// TwinCAT 3 PLC project PLC_Tool_Magazine_8xx
// ProgramVersion: 3.1.4026.20
// libraries:
//   Tc2_Drive, * (Beckhoff Automation GmbH)
//   Tc2_Math, * (Beckhoff Automation GmbH)
//   Tc2_MC2, * (Beckhoff Automation GmbH)
//   Tc2_MC2_Drive, * (Beckhoff Automation GmbH)
//   Tc2_Standard, * (Beckhoff Automation GmbH)
//   Tc2_System, * (Beckhoff Automation GmbH)
//   Tc2_Utilities, * (Beckhoff Automation GmbH)
//   Tc3_EventLogger, * (Beckhoff Automation GmbH)
//   Tc3_IoLink, * (Beckhoff Automation GmbH)
//   Tc3_Module, * (Beckhoff Automation GmbH)
// project tree:
//   01_General %28MAIN%29/01_DUTs/01_ENUM/ ENUM_VarType.TcDUT (not stored)
//   01_General %28MAIN%29/01_DUTs/02_ST/ ST_Array_Data.TcDUT (not stored), ST_Miscellaneous.TcDUT (not stored), ST_Pointer_Data.TcDUT (not stored)
//   01_General %28MAIN%29/02_GVLs/ GV_General.TcGVL (not stored), GV_IO.TcGVL (not stored)
//   01_General %28MAIN%29/03_POUs/01_PRGs/ PRG_Backup.TcPOU (not stored), PRG_FirstCycle.TcPOU (not stored), PRG_Main.TcPOU (not stored), PRG_SavePersistentData.TcPOU (not stored)
//   01_General %28MAIN%29/03_POUs/02_FBs/ FB_ArrayToolLocation_Reverse.TcPOU (not stored), FB_BackupExport.TcPOU (not stored), FB_BackupImport.TcPOU (not stored), FB_Blink.TcPOU (not stored)
//   02_Events/01_DUTs/02_ST/ ST_Alarm.TcDUT, ST_Event_Group.TcDUT, ST_Message.TcDUT
//   02_Events/02_GVLs/ GV_Events.TcGVL
//   02_Events/03_POUs/02_FBs/ FB_Event_Group_Number_Assignement.TcPOU, FB_Event_HMI.TcPOU, FB_Init_Call_Events.TcPOU, FB_Init_Events.TcPOU
//   03_Operating_Mode/01_DUTs/01_ENUM/ ENUM_OpMode.TcDUT
//   03_Operating_Mode/02_GVLs/ GV_OpMode.TcGVL
//   03_Operating_Mode/03_POUs/01_PRGs/ PRG_OpMode.TcPOU
//   04_Lamps_Lights/03_POUs/01_PRGs/ PRG_Lamps_Lights.TcPOU
//   05_Fans/01_DUTs/01_ENUM/ ENUM_Fan_Type.TcDUT
//   05_Fans/01_DUTs/02_ST/ ST_Fan.TcDUT
//   05_Fans/02_GVLs/ GV_Fans.TcGVL
//   05_Fans/03_POUs/01_PRGs/ PRG_Fans.TcPOU
//   05_Fans/03_POUs/02_FBs/ FB_Fan.TcPOU
//   06_Doors/01_DUTs/01_ENUM/ ENUM_Door_Type.TcDUT
//   06_Doors/01_DUTs/02_ST/ ST_Door.TcDUT
//   06_Doors/02_GVLs/ GV_Doors.TcGVL
//   06_Doors/03_POUs/01_PRGs/ PRG_Doors.TcPOU
//   06_Doors/03_POUs/02_FBs/ FB_Door.TcPOU
//   07_Cyltronic/01_DUTs/01_ENUM/ ENUM_Cyltronic_Type.TcDUT, teCTCBrakeMode.TcTLEO, teCTCConfigStep.TcDUT, teCTCDeviceStatus.TcTLEO, teCTCEvent.TcTLEO, teCTCGDSStep.TcDUT, teCTCHomeMode.TcTLEO, teCTCStep.TcTLEO, teCTCWarningID.TcTLEO
//   07_Cyltronic/01_DUTs/02_ST/ ST_Cyltronic.TcDUT, tstCTCConfiguration.TcDUT, tstCTCConfigVariable.TcDUT, tstCTCDeviceStatus.TcDUT, tstCTCEvent.TcDUT, tstCTCInternalCommands.TcDUT, tstCTCParameters.TcDUT, tstCTCProcessDataIn.TcDUT, tstCTCProcessDataOut.TcDUT, tstCTCStatusBits.TcDUT
//   07_Cyltronic/01_DUTs/03_Union/ tuReal.TcDUT
//   07_Cyltronic/02_GVLs/ CTC_CONSTANTS.TcGVL, GV_Cyltronic.TcGVL
//   07_Cyltronic/03_POUs/01_PRGs/ PRG_Cyltronic.TcPOU
//   07_Cyltronic/03_POUs/02_FBs/ FB_CTC_Basic.TcPOU, FB_CTC_GetDeviceStatus.TcPOU, FB_CTC_PlcOpen.TcPOU, FB_CTC_ReadWriteConfig.TcPOU, FB_Cyltronic.TcPOU
//   08_Cycle/01_DUTs/01_ENUM/ ENUM_Cycle_Action.TcDUT, ENUM_Cycle_Step.TcDUT, ENUM_Cycle_Type.TcDUT
//   08_Cycle/02_GVLs/ GV_Cycle.TcGVL
//   08_Cycle/03_POUs/01_PRGs/ PRG_Cycle_AlarmsMessages.TcPOU, PRG_Cycle.TcPOU
//   08_Cycle/03_POUs/02_FBs/ FB_01_Action_PickToolMagazine.TcPOU, FB_05_Action_PlaceToolMagazine.TcPOU, FB_10_Action_ToolMagazineCheckOne.TcPOU, FB_200_Action_HomePosition.TcPOU, FB_202_Action_PickPlaceToolMag.TcPOU, FB_20_Action_Initialization.TcPOU, FB_03_Action_TransferArmCnc.TcPOU, FB_02_Action_TransferManipulatorToArm.TcPOU, FB_04_Action_TransferArmToManipulator.TcPOU, FB_11_Action_ToolMagazineCheckAll.TcPOU
//   09_Tool_Magazine/01_DUTs/01_ENUM/ ENUM_Gripper_Mode.TcDUT, ENUM_Position_Axis.TcDUT, ENUM_Position_Magazine.TcDUT, ENUM_Tool_Type.TcDUT, ENUM_Tunnel_Mode.TcDUT
//   09_Tool_Magazine/01_DUTs/02_ST/ ST_Changing_Arm.TcDUT, ST_Changing_Arm_Gripper.TcDUT, ST_Manipulator_Head.TcDUT, ST_Tool_Corrector_M.TcDUT, ST_Tool_Corrector_T.TcDUT, ST_Tool_Name.TcDUT, ST_Tool_Parameters.TcDUT, ST_Tool_Location.TcDUT
//   09_Tool_Magazine/02_GVLs/ GV_Tool_Magazine.TcGVL
//   09_Tool_Magazine/03_POUs/01_PRGs/ PRG_Tool_Magazine_Type1_Refresh.TcPOU, PRG_Tool_Magazine_Type1.TcPOU
//   09_Tool_Magazine/03_POUs/02_FBs/ FB_Manipulator_Breakage.TcPOU, FB_Manipulator_Gripper.TcPOU, FB_Manipulator_Tunnel.TcPOU, FB_Manipulator_Tunnel_5.TcPOU, FB_Manipulator_Tunnel_2.TcPOU
//   10_Axes/01_DUTs/01_ENUM/ ENUM_Axis_Mode.TcDUT, ENUM_Axis_Status.TcDUT, ENUM_Axis_Select.TcDUT, ENUM_Handwheel_Incr_Select.TcDUT, ENUM_Jog_Direction.TcDUT, ENUM_Jog_Mode.TcDUT
//   10_Axes/01_DUTs/02_ST/ ST_Axis.TcDUT, ST_Beckhoff_Drive_AX8206.TcDUT, ST_Handwheel.TcDUT
//   10_Axes/02_GVLs/ GV_Axes.TcGVL, GV_Handwheel.TcGVL
//   10_Axes/03_POUs/01_PRGs/ PRG_Handwheel.TcPOU, PRG_Axis.TcPOU
//   10_Axes/03_POUs/02_FBs/ FB_Axis.TcPOU, FB_Handwheel.TcPOU, FB_Handwheel_2.TcPOU
//   11_CNC/01_DUTs/01_ENUM/ ENUM_CNC_Type.TcDUT
//   11_CNC/01_DUTs/02_ST/ ST_CNC_Fanuc_Data.TcDUT, ST_CNC_Fanuc_Focas_Data.TcDUT, ST_CNC_Heidenhain_Exchange_In_1.TcDUT, ST_CNC_Heidenhain_Exchange_Out_1.TcDUT, ST_CNC_Heidenhain_Data.TcDUT, ST_CNC_Fanuc_Exchange_In_1.TcDUT, ST_CNC_Fanuc_Exchange_Out_1.TcDUT, ST_Spindle.TcDUT
//   11_CNC/02_GVLs/ GV_CNC.TcGVL
//   11_CNC/03_POUs/01_PRGs/ PRG_CNC.TcPOU
//   11_CNC/03_POUs/02_FBs/ FB_CNC_Fanuc.TcPOU, FB_CNC_Heidenhain.TcPOU
//   12_Focas/01_DUTs/02_ST/ St_Write_Focas.TcDUT, ST_Focas_To_Magazine.TcDUT, St_Read_Focas.TcDUT, ST_Magazine_To_Focas.TcDUT
//   12_Focas/02_GVLs/ GV_Focas.TcGVL
//   12_Focas/03_POUs/01_PRGs/ PRG_Focas.TcPOU
//   12_Focas/03_POUs/02_FBs/ FB_ConnectionFocas.TcPOU, FB_ReadFocas.TcPOU, FB_WriteFocas.TcPOU
//   13_HMI/01_DUTs/01_ENUM/ ENUM_User_Level.TcDUT
//   13_HMI/01_DUTs/02_ST/ ST_HMI_Axes.TcDUT, ST_HMI_Backup.TcDUT, ST_HMI_Cycle.TcDUT, ST_HMI_Cyltronic.TcDUT, ST_HMI_Doors.TcDUT, ST_HMI_Footer.TcDUT, ST_HMI_Header.TcDUT, ST_HMI_Lamps_Lights.TcDUT, ST_HMI_Magazine_Check.TcDUT, ST_HMI_Magazine_Settings.TcDUT, ST_HMI_Magazine_Teach.TcDUT, ST_HMI_Manipulator_Gripper.TcDUT, ST_HMI_Manipulator_Breakage.TcDUT, ST_HMI_Manipulator_Tunnel.TcDUT, ST_HMI_Pick_Tool_Magazine.TcDUT, ST_HMI_Transfer_ManipulatorToArm.TcDUT, ST_HMI_Screen_Home.TcDUT, ST_HMI_Transfer_ArmCnc.TcDUT, ST_HMI_Transfer_ArmToManipulator.TcDUT
//   13_HMI/02_GVLs/ GV_HMI.TcGVL
//   13_HMI/03_POUs/01_PRGs/ PRG_HMI.TcPOU
//   14_Log/01_DUTs/01_ENUM/ ENUM_Log_File_Management.TcDUT, ENUM_Log_Type.TcDUT
//   14_Log/01_DUTs/02_ST/ ST_Log.TcDUT, ST_Log_Data.TcDUT
//   14_Log/02_GVLs/ GV_Log.TcGVL
//   14_Log/03_POUs/01_PRGs/ PRG_Log.TcPOU, PRG_Log_WM.TcPOU
//   14_Log/03_POUs/02_FBs/ FB_Log.TcPOU, FB_Write_DataToFile.TcPOU, sTime.TcPOU
//   / PlcTask.TcTTO
// real-time tasks:
//   TASK PlcTask: cycle T#8ms, priority 20, ADS port 350
// motion (NC):
//   TASK NC-Task 1 SAF: cycle T#2ms, priority 4, ADS port 501
//   TASK NC-Task 1 SVB: cycle T#10ms, priority 8, ADS port 511
//   AXIS A64.1 - Axis Z (id 1)
//     Dynamic: Acceleration=768, Deceleration=768, Jerk=1536
//     Velo: RefSearch=16.34233, RefSync=16.34233, SlowManual=81.71165, FastManual=490.2699, Fast=1634.233, Maximum=384
//     OtherSettings: AllowMotionCmdToSlave=true, PulseDistancePos=1, PulseDistanceNeg=1
//     encoder EncType=19
//       EncPara: ScaleFactorNumerator=20, ScaleFactorDenominator=1048576, MaxCount=#xffffffff
//         SoftEndMinControl: Enable=true, Range=-0.1
//         SoftEndMaxControl: Enable=true, Range=1152.1
//     drive DrvType=16
//       DrvPara: MaxCount=#xffffffff, DriveControlDWord=#x00020100
//         Analog: VeloReferenz=422, VeloScale=71.5255737304688, TorqueSetpointScale=10, ScaleFactorActTorque=0.1
//         TimeComp: TaskDelayCycles=1
//     controller CtrType=1
//       CtrPara: PriorControlFactor=1
//         PosDiffControl: Range=0.2
//         Observer: BandWidth=20
//   AXIS A64.1 - Axis X (id 2)
//     Dynamic: Acceleration=7000, Deceleration=7000, Jerk=100000
//     Velo: RefSearch=10, RefSync=10, SlowManual=25, FastManual=50, Fast=2850, Maximum=697
//     OtherSettings: AllowMotionCmdToSlave=true, PulseDistancePos=1, PulseDistanceNeg=1
//     encoder EncType=19
//       EncPara: ScaleFactorNumerator=20, ScaleFactorDenominator=1048576, MaxCount=#xffffffff
//         SoftEndMinControl: Enable=true, Range=-0.1
//         SoftEndMaxControl: Enable=true, Range=684.6
//     drive DrvType=16
//       DrvPara: MaxCount=#xffffffff, DriveControlDWord=#x00020100
//         Analog: VeloReferenz=3135, VeloScale=71.5255737304688, TorqueSetpointScale=10, ScaleFactorActTorque=0.1
//         TimeComp: TaskDelayCycles=1
//     controller CtrType=1
//       CtrPara: PriorControlFactor=1
//         Observer: BandWidth=20
//   AXIS A64.2 - Axis Y (id 3)
//     Dynamic: Acceleration=6390, Deceleration=6390, Jerk=220000
//     Velo: RefSearch=10, RefSync=10, SlowManual=25, FastManual=50, Fast=6268.29, Maximum=169
//     OtherSettings: AllowMotionCmdToSlave=true, PulseDistancePos=1, PulseDistanceNeg=1
//     encoder EncType=19
//       EncPara: ScaleFactorNumerator=43.988, ScaleFactorDenominator=1048576, MaxCount=#xffffffff
//         SoftEndMinControl: Enable=true, Range=-0.1
//         SoftEndMaxControl: Enable=true, Range=72.6
//     drive DrvType=16
//       DrvPara: MaxCount=#xffffffff, DriveControlDWord=#x00020100
//         Analog: VeloReferenz=6895.119, VeloScale=71.5255737304688, TorqueSetpointScale=10, ScaleFactorActTorque=0.1
//         TimeComp: TaskDelayCycles=1
//     controller CtrType=1
//       CtrPara: PriorControlFactor=1
//         Observer: BandWidth=20
//   AXIS A64.2 - Axis Arm (id 4)
//     Dynamic: Acceleration=3000, Deceleration=3000, Jerk=155000
//     Velo: RefSearch=10, RefSync=10, SlowManual=25, FastManual=50, Fast=2280, Maximum=641
//     OtherSettings: AllowMotionCmdToSlave=true, PulseDistancePos=1, PulseDistanceNeg=1
//     encoder EncType=19
//       EncPara: ScaleFactorNumerator=16, ScaleFactorDenominator=1048576, MaxCount=#xffffffff
//         SoftEndMinControl: Enable=true, Range=-0.1
//         SoftEndMaxControl: Enable=true, Range=332.1
//     drive DrvType=16
//       DrvPara: MaxCount=#xffffffff, DriveControlDWord=#x00020100
//         Analog: VeloReferenz=700, VeloScale=71.5255737304688, TorqueSetpointScale=10, ScaleFactorActTorque=0.1
//         TimeComp: TaskDelayCycles=1
//     controller CtrType=1
//       CtrPara: PriorControlFactor=1
//         Observer: BandWidth=20
// I/O:
//   DEVICE Device 2 (EtherCAT), AmsNetId 10.1.176.55.3.1
//     U101.1 (EK1200) [EK1200-5000 EtherCAT Power supply (2A E-Bus)]
//       I271 (EL1809) [EL1809 16Ch. Dig. Input 24V, 3ms]
//       IO273 (EL8601-8411) [EL8601-8411 12Ch. Multi-interface, 8x DI, 1x CNT, 4x DO, 2x PWM, 1x AI, 1x AO, 1x ENC AB]
//         modules: SlotGroup 1 (CNT_2xDI), SlotGroup 1 (CNT_2xDI), SlotGroup 1 (CNT_2xDI), SlotGroup 1 (CNT_2xDI), SlotGroup 2 (DI_4x), SlotGroup 2 (DI_4x), SlotGroup 2 (DI_4x), SlotGroup 2 (DI_4x), SlotGroup 3 (PWM_OUT_DO), SlotGroup 3 (PWM_OUT_DO), SlotGroup 4 (AI_1xV), SlotGroup 5 (AO_1xV)
//       O275 (EL2809) [EL2809 16Ch. Dig. Output 24V, 0.5A]
//       A277 (EL6224) [EL6224 (IO Link Master)]
//       A270.1 [EK1122 2 port EtherCAT junction]
//         A64 (AX8620-0000-0105) [AX8620-0000-0105]
//           A64.1 (AX8206-0200-0107) [AX8206-0200-0107 (2Ch. 6A servo axis, safe-motion)]
//             modules: Device, Device, Device, Device, Device, Device, Device, Device, Device, Device, Device (Safety), Device, Device, Device, Device, Device, Device, Device, Device, Device, Device, Device, Device, Device, Device, Device, Device, Device, Device, Device, Device, Ch A, Ch A, Ch A, Ch A, Ch A, Ch A, Ch A, Ch A, Ch A, Ch A, Ch A, Ch A, Ch A, Ch A, Ch A, Ch A, Ch A, Ch A, Ch A, Ch A, Ch A, Ch A, Ch A, Ch A, Ch A, Ch A, Ch A, Ch A, Ch A, Ch A, Ch B, Ch B, Ch B, Ch B, Ch B, Ch B, Ch B, Ch B, Ch B, Ch B, Ch B, Ch B, Ch B, Ch B, Ch B, Ch B, Ch B, Ch B, Ch B, Ch B, Ch B, Ch B, Ch B, Ch B, Ch B, Ch B, Ch B
//             startup 12992:1 := 414D383032312D78427831 // Ch A SynchronousMotor parameters / Configured motor type
//             startup 24768:0 := FEFF // Ch A Interpolation sub mode select
//             startup 13000:5 := 0200 // Ch A SynchronousMotor thermal model / Reaction
//             startup 13000:6 := 0000C841 // Ch A SynchronousMotor thermal model / Partial fraction factor
//             startup 12992:12 := 0000FA45 // Ch A SynchronousMotor parameters / Motor rated speed
//             startup 12992:13 := C9E5FF3E // Ch A SynchronousMotor parameters / Motor rated torque
//             startup 24694:0 := F4010000 // Ch A Motor standstill torque
//             startup 24800:0 := D007 // Ch A Positive torque/force limit value
//             startup 24801:0 := D007 // Ch A Negative torque/force limit value
//             startup 12288:6 := 4158383230362D303230302D30303030 // Ch A AxisMain parameters / Configured drive type
//             startup 12867:1 := 9A99593F // Ch A TorqueControl parameters / Configured channel rated current
//             startup 12867:2 := 33332340 // Ch A TorqueControl parameters / Configured channel peak current
//             startup 12867:7 := 77BE1F40 // Ch A TorqueControl parameters / Iuvw max sum
//             startup 24672:0 := 08 // Ch A Modes of operation
//             startup 13023:0 := 0000 // Ch A SynchronousMotor control mode
//             startup 12998:1 := C09D7E3D // Ch A SynchronousMotor commutation monitoring parameters / Speed threshold
//             startup 12864:1 := 0D4D7043 // Ch A TorqueControl parameters mappable / Torque control proportional gain q
//             startup 12864:2 := 8A0E7C39 // Ch A TorqueControl parameters mappable / Torque control integral action time q
//             startup 12608:1 := 870B223C // Ch A VelocityControl parameters mappable / Velocity control proportional gain
//             startup 12608:2 := 6F12033C // Ch A VelocityControl parameters mappable / Velocity control integral action time
//             startup 12608:3 := 00980546 // Ch A VelocityControl parameters mappable / Bipolar velocity limit value
//             startup 12992:15 := 0100 // Ch A SynchronousMotor parameters / Motor temperature sensor connection
//             startup 12611:4 := 0400 // Ch A VelocityControl observer / Observer type
//             startup 24672:0 := 08 // Ch A Modes of operation
//             startup 12296:2 := 00 // Ch A AxisMain parameters encoder direction / Primary encoder direction
//             startup 14016:1 := 414D383031332D78447830 // Ch B SynchronousMotor parameters / Configured motor type
//             startup 26816:0 := FEFF // Ch B Interpolation sub mode select
//             startup 14024:5 := 0200 // Ch B SynchronousMotor thermal model / Reaction
//             startup 14024:6 := 0000C841 // Ch B SynchronousMotor thermal model / Partial fraction factor
//             startup 14016:12 := 0000FA45 // Ch B SynchronousMotor parameters / Motor rated speed
//             startup 14016:13 := FCA9D13E // Ch B SynchronousMotor parameters / Motor rated torque
//             startup 26742:0 := 08020000 // Ch B Motor standstill torque
//             startup 26848:0 := D007 // Ch B Positive torque/force limit value
//             startup 26849:0 := D007 // Ch B Negative torque/force limit value
//             startup 13312:6 := 4158383230362D303230302D30303030 // Ch B AxisMain parameters / Configured drive type
//             startup 13891:1 := 3333D33F // Ch B TorqueControl parameters / Configured channel rated current
//             startup 13891:2 := 66669E40 // Ch B TorqueControl parameters / Configured channel peak current
//             startup 13891:7 := 77BE1F40 // Ch B TorqueControl parameters / Iuvw max sum
//             startup 26720:0 := 08 // Ch B Modes of operation
//             startup 14047:0 := 0000 // Ch B SynchronousMotor control mode
//             startup 14022:1 := 0AD7A33D // Ch B SynchronousMotor commutation monitoring parameters / Speed threshold
//             startup 13888:1 := F01D0142 // Ch B TorqueControl parameters mappable / Torque control proportional gain q
//             startup 13888:2 := 8A0E7C39 // Ch B TorqueControl parameters mappable / Torque control integral action time q
//             startup 13632:1 := 102E5D3B // Ch B VelocityControl parameters mappable / Velocity control proportional gain
//             startup 13632:2 := 6F12033C // Ch B VelocityControl parameters mappable / Velocity control integral action time
//             startup 13632:3 := 00980546 // Ch B VelocityControl parameters mappable / Bipolar velocity limit value
//             startup 13635:4 := 0400 // Ch B VelocityControl observer / Observer type
//             startup 26720:0 := 08 // Ch B Modes of operation
//             startup 13320:2 := 00 // Ch B AxisMain parameters encoder direction / Primary encoder direction
//           A64.2 (AX8206-0200-0107) [AX8206-0200-0107 (2Ch. 6A servo axis, safe-motion)]
//             modules: Device, Device, Device, Device, Device, Device, Device, Device, Device, Device, Device (Safety), Device, Device, Device, Device, Device, Device, Device, Device, Device, Device, Device, Device, Device, Device, Device, Device, Device, Device, Device, Device, Ch A, Ch A, Ch A, Ch A, Ch A, Ch A, Ch A, Ch A, Ch A, Ch A, Ch A, Ch A, Ch A, Ch A, Ch A, Ch A, Ch A, Ch A, Ch A, Ch A, Ch A, Ch A, Ch A, Ch A, Ch A, Ch A, Ch A, Ch B, Ch B, Ch B, Ch B, Ch B, Ch B, Ch B, Ch B, Ch B, Ch B, Ch B, Ch B, Ch B, Ch B, Ch B, Ch B, Ch B, Ch B, Ch B, Ch B, Ch B, Ch B, Ch B, Ch B, Ch B, Ch B, Ch B
//             startup 12992:1 := 414D383031322D78437830 // Ch A SynchronousMotor parameters / Configured motor type
//             startup 24768:0 := FEFF // Ch A Interpolation sub mode select
//             startup 13000:5 := 0200 // Ch A SynchronousMotor thermal model / Reaction
//             startup 13000:6 := 0000C841 // Ch A SynchronousMotor thermal model / Partial fraction factor
//             startup 12992:12 := 0000FA45 // Ch A SynchronousMotor parameters / Motor rated speed
//             startup 12992:13 := A167B33E // Ch A SynchronousMotor parameters / Motor rated torque
//             startup 24694:0 := 7C010000 // Ch A Motor standstill torque
//             startup 24800:0 := D007 // Ch A Positive torque/force limit value
//             startup 24801:0 := D007 // Ch A Negative torque/force limit value
//             startup 12288:6 := 4158383230362D303230302D30303030 // Ch A AxisMain parameters / Configured drive type
//             startup 12867:1 := 6666A63F // Ch A TorqueControl parameters / Configured channel rated current
//             startup 12867:2 := 9A997940 // Ch A TorqueControl parameters / Configured channel peak current
//             startup 12867:7 := 77BE1F40 // Ch A TorqueControl parameters / Iuvw max sum
//             startup 24672:0 := 08 // Ch A Modes of operation
//             startup 13023:0 := 0000 // Ch A SynchronousMotor control mode
//             startup 12998:1 := 0AD7A33D // Ch A SynchronousMotor commutation monitoring parameters / Speed threshold
//             startup 12864:1 := EEA21642 // Ch A TorqueControl parameters mappable / Torque control proportional gain q
//             startup 12864:2 := 8A0E7C39 // Ch A TorqueControl parameters mappable / Torque control integral action time q
//             startup 12608:1 := 696D233B // Ch A VelocityControl parameters mappable / Velocity control proportional gain
//             startup 12608:2 := 6F12033C // Ch A VelocityControl parameters mappable / Velocity control integral action time
//             startup 12608:3 := 00980546 // Ch A VelocityControl parameters mappable / Bipolar velocity limit value
//             startup 12611:4 := 0400 // Ch A VelocityControl observer / Observer type
//             startup 24672:0 := 08 // Ch A Modes of operation
//             startup 12296:2 := 00 // Ch A AxisMain parameters encoder direction / Primary encoder direction
//             startup 14016:1 := 414D383031332D78447830 // Ch B SynchronousMotor parameters / Configured motor type
//             startup 26816:0 := FEFF // Ch B Interpolation sub mode select
//             startup 14024:5 := 0200 // Ch B SynchronousMotor thermal model / Reaction
//             startup 14024:6 := 0000C841 // Ch B SynchronousMotor thermal model / Partial fraction factor
//             startup 14016:12 := 0000FA45 // Ch B SynchronousMotor parameters / Motor rated speed
//             startup 14016:13 := FCA9D13E // Ch B SynchronousMotor parameters / Motor rated torque
//             startup 26742:0 := 08020000 // Ch B Motor standstill torque
//             startup 26848:0 := D007 // Ch B Positive torque/force limit value
//             startup 26849:0 := D007 // Ch B Negative torque/force limit value
//             startup 13312:6 := 4158383230362D303230302D30303030 // Ch B AxisMain parameters / Configured drive type
//             startup 13891:1 := 3333D33F // Ch B TorqueControl parameters / Configured channel rated current
//             startup 13891:2 := 66669E40 // Ch B TorqueControl parameters / Configured channel peak current
//             startup 13891:7 := 77BE1F40 // Ch B TorqueControl parameters / Iuvw max sum
//             startup 26720:0 := 08 // Ch B Modes of operation
//             startup 14047:0 := 0000 // Ch B SynchronousMotor control mode
//             startup 14022:1 := 0AD7A33D // Ch B SynchronousMotor commutation monitoring parameters / Speed threshold
//             startup 13888:1 := F01D0142 // Ch B TorqueControl parameters mappable / Torque control proportional gain q
//             startup 13888:2 := 8A0E7C39 // Ch B TorqueControl parameters mappable / Torque control integral action time q
//             startup 13632:1 := 102E5D3B // Ch B VelocityControl parameters mappable / Velocity control proportional gain
//             startup 13632:2 := 6F12033C // Ch B VelocityControl parameters mappable / Velocity control integral action time
//             startup 13632:3 := 00980546 // Ch B VelocityControl parameters mappable / Bipolar velocity limit value
//             startup 13635:4 := 0400 // Ch B VelocityControl observer / Observer type
//             startup 26720:0 := 08 // Ch B Modes of operation
//             startup 13320:2 := 00 // Ch B AxisMain parameters encoder direction / Primary encoder direction
//       U270-T (EL9011) [EL9011 End Terminal]
//   DEVICE Device 1 (Profinet Device CCAT (RT)), AmsNetId 10.1.176.55.2.1
//     toolmagazine000 [Beckhoff Automation CX2xx0-B930 PROFINET IO Device with I/Os; V2.43; PROFIenergy supported CX2xx0-B930]
//       modules: Term 1 (DAP Module), I1 (8 Byte Input), I2 (4 Word Input), I3 (16 Byte Input), O1 (8 Byte Output), O2 (4 Word Output), O3 (16 Byte Output)
// variable links:
//   Device 2 (EtherCAT) <-> Device 2 (EtherCAT)/U101.1 (EK1200)/A270.1/A64 (AX8620-0000-0105)
//     U101.1 (EK1200)/A270.1/A64 (AX8620-0000-0105)/A64.1 (AX8206-0200-0107)/Device/DeviceMain Outputs/Power supply controlword <-> PSM Controlword for axis/Controlword for axis
//     U101.1 (EK1200)/A270.1/A64 (AX8620-0000-0105)/A64.2 (AX8206-0200-0107)/Device/DeviceMain Outputs/Power supply controlword <-> PSM Controlword for axis/Controlword for axis
//   PLC_Tool_Magazine_8xx/PLC_Tool_Magazine_8xx Instance <-> Device 1 (Profinet Device CCAT (RT))/toolmagazine000
//     PlcTask Inputs/GV_CNC.stFanucData.stCncMagazine.byi{0..5} <-> API/O1 (8 Byte Output)/Subterm 8 (8 Byte Output)/Inputs/1 Byte Output[{0..5}]  (6 links)
//     PlcTask Inputs/GV_CNC.stFanucData.stCncMagazine.byiResevrve{16..31} <-> API/O3 (16 Byte Output)/Subterm 10 (16 Byte Output)/Inputs/1 Byte Output[{0..15}]  (16 links)
//     PlcTask Inputs/GV_CNC.stFanucData.stCncMagazine.byiSpindleToolType <-> API/O1 (8 Byte Output)/Subterm 8 (8 Byte Output)/Inputs/1 Byte Output[6]
//     PlcTask Inputs/GV_CNC.stFanucData.stCncMagazine.byiToolToLoadType <-> API/O1 (8 Byte Output)/Subterm 8 (8 Byte Output)/Inputs/1 Byte Output[7]
//     PlcTask Inputs/GV_CNC.stFanucData.stCncMagazine.wiPT100ArmorStatus <-> API/O2 (4 Word Output)/Subterm 9 (4 Word Output)/Inputs/1 Word Output[2]
//     PlcTask Inputs/GV_CNC.stFanucData.stCncMagazine.wiPT100ArmorValue <-> API/O2 (4 Word Output)/Subterm 9 (4 Word Output)/Inputs/1 Word Output[3]
//     PlcTask Inputs/GV_CNC.stFanucData.stCncMagazine.wiSpindleToolLocation <-> API/O2 (4 Word Output)/Subterm 9 (4 Word Output)/Inputs/1 Word Output[0]
//     PlcTask Inputs/GV_CNC.stFanucData.stCncMagazine.wiToolToLoadLocation <-> API/O2 (4 Word Output)/Subterm 9 (4 Word Output)/Inputs/1 Word Output[1]
//     PlcTask Outputs/GV_CNC.stFanucData.stMagazineCNC.byo{0..5} <-> API/I1 (8 Byte Input)/Subterm 5 (8 Byte Input)/Outputs/1 Byte Input[{0..5}]  (6 links)
//     PlcTask Outputs/GV_CNC.stFanucData.stMagazineCNC.byoResevrve16 <-> API/I3 (16 Byte Input)/Subterm 7 (16 Byte Input)/Outputs/1 Byte Input[0]
//     PlcTask Outputs/GV_CNC.stFanucData.stMagazineCNC.byoResevrve17 <-> API/I3 (16 Byte Input)/Subterm 7 (16 Byte Input)/Outputs/1 Byte Input[1]
//     PlcTask Outputs/GV_CNC.stFanucData.stMagazineCNC.byoResevrve18 <-> API/I3 (16 Byte Input)/Subterm 7 (16 Byte Input)/Outputs/1 Byte Input[2]
//     PlcTask Outputs/GV_CNC.stFanucData.stMagazineCNC.byoResevrve19 <-> API/I3 (16 Byte Input)/Subterm 7 (16 Byte Input)/Outputs/1 Byte Input[3]
//     PlcTask Outputs/GV_CNC.stFanucData.stMagazineCNC.byoResevrve20 <-> API/I3 (16 Byte Input)/Subterm 7 (16 Byte Input)/Outputs/1 Byte Input[4]
//     PlcTask Outputs/GV_CNC.stFanucData.stMagazineCNC.byoResevrve21 <-> API/I3 (16 Byte Input)/Subterm 7 (16 Byte Input)/Outputs/1 Byte Input[5]
//     PlcTask Outputs/GV_CNC.stFanucData.stMagazineCNC.byoResevrve22 <-> API/I3 (16 Byte Input)/Subterm 7 (16 Byte Input)/Outputs/1 Byte Input[6]
//     PlcTask Outputs/GV_CNC.stFanucData.stMagazineCNC.byoResevrve23 <-> API/I3 (16 Byte Input)/Subterm 7 (16 Byte Input)/Outputs/1 Byte Input[7]
//     PlcTask Outputs/GV_CNC.stFanucData.stMagazineCNC.byoResevrve24 <-> API/I3 (16 Byte Input)/Subterm 7 (16 Byte Input)/Outputs/1 Byte Input[8]
//     PlcTask Outputs/GV_CNC.stFanucData.stMagazineCNC.byoResevrve25 <-> API/I3 (16 Byte Input)/Subterm 7 (16 Byte Input)/Outputs/1 Byte Input[9]
//     PlcTask Outputs/GV_CNC.stFanucData.stMagazineCNC.byoResevrve26 <-> API/I3 (16 Byte Input)/Subterm 7 (16 Byte Input)/Outputs/1 Byte Input[10]
//     PlcTask Outputs/GV_CNC.stFanucData.stMagazineCNC.byoResevrve27 <-> API/I3 (16 Byte Input)/Subterm 7 (16 Byte Input)/Outputs/1 Byte Input[11]
//     PlcTask Outputs/GV_CNC.stFanucData.stMagazineCNC.byoResevrve28 <-> API/I3 (16 Byte Input)/Subterm 7 (16 Byte Input)/Outputs/1 Byte Input[12]
//     PlcTask Outputs/GV_CNC.stFanucData.stMagazineCNC.byoResevrve29 <-> API/I3 (16 Byte Input)/Subterm 7 (16 Byte Input)/Outputs/1 Byte Input[13]
//     PlcTask Outputs/GV_CNC.stFanucData.stMagazineCNC.byoResevrve30 <-> API/I3 (16 Byte Input)/Subterm 7 (16 Byte Input)/Outputs/1 Byte Input[14]
//     PlcTask Outputs/GV_CNC.stFanucData.stMagazineCNC.byoResevrve31 <-> API/I3 (16 Byte Input)/Subterm 7 (16 Byte Input)/Outputs/1 Byte Input[15]
//     PlcTask Outputs/GV_CNC.stFanucData.stMagazineCNC.byoResevrve6 <-> API/I1 (8 Byte Input)/Subterm 5 (8 Byte Input)/Outputs/1 Byte Input[6]
//     PlcTask Outputs/GV_CNC.stFanucData.stMagazineCNC.byoResevrve7 <-> API/I1 (8 Byte Input)/Subterm 5 (8 Byte Input)/Outputs/1 Byte Input[7]
//     PlcTask Outputs/GV_CNC.stFanucData.stMagazineCNC.woReserve10 <-> API/I2 (4 Word Input)/Subterm 6 (4 Word Input)/Outputs/1 Word Input[1]
//     PlcTask Outputs/GV_CNC.stFanucData.stMagazineCNC.woReserve8 <-> API/I2 (4 Word Input)/Subterm 6 (4 Word Input)/Outputs/1 Word Input[0]
//     PlcTask Outputs/GV_CNC.stFanucData.stMagazineCNC.woResevrve12 <-> API/I2 (4 Word Input)/Subterm 6 (4 Word Input)/Outputs/1 Word Input[2]
//     PlcTask Outputs/GV_CNC.stFanucData.stMagazineCNC.woResevrve14 <-> API/I2 (4 Word Input)/Subterm 6 (4 Word Input)/Outputs/1 Word Input[3]
//   PLC_Tool_Magazine_8xx/PLC_Tool_Magazine_8xx Instance <-> Device 2 (EtherCAT)/U101.1 (EK1200)/A277 (EL6224)
//     PlcTask Inputs/GV_Cyltronic.aId[1].aProcessDataInRaw <-> IO-Link Port1_in/Port1: process data
//     PlcTask Inputs/GV_Tool_Magazine.uiBreakageSensor <-> IO-Link Port2/Port2: process data
//     PlcTask Outputs/GV_Cyltronic.aId[1].aProcessDataOutRaw <-> IO-Link Port1_out/Port1: process data
//   PLC_Tool_Magazine_8xx/PLC_Tool_Magazine_8xx Instance <-> Device 2 (EtherCAT)/U101.1 (EK1200)/I271 (EL1809)
//     PlcTask Inputs/GV_IO.diButtonUnlockMagazineDoor <-> Channel 14/Input
//     PlcTask Inputs/GV_IO.diEmergencyStop <-> Channel 1/Input
//     PlcTask Inputs/GV_IO.diHandwheelAxisSelectorB0 <-> Channel 2/Input
//     PlcTask Inputs/GV_IO.diHandwheelAxisSelectorB1 <-> Channel 3/Input
//     PlcTask Inputs/GV_IO.diHandwheelAxisSelectorB2 <-> Channel 4/Input
//     PlcTask Inputs/GV_IO.diIntermediateDoorNotClosed <-> Channel 10/Input
//     PlcTask Inputs/GV_IO.diMagazineDoorOpen <-> Channel 15/Input
//     PlcTask Inputs/GV_IO.diReserve27111 <-> Channel 11/Input
//     PlcTask Inputs/GV_IO.diReserve2716 <-> Channel 6/Input
//     PlcTask Inputs/GV_IO.diReserve2717 <-> Channel 7/Input
//     PlcTask Inputs/GV_IO.diSafetyAreaMagazineOk <-> Channel 9/Input
//     PlcTask Inputs/GV_IO.diSafetyRelayIntermediateDoor <-> Channel 16/Input
//     PlcTask Inputs/GV_IO.diSafetyRelayMagazineDoor <-> Channel 5/Input
//     PlcTask Inputs/GV_IO.diToolPresenceArmGripper1 <-> Channel 12/Input
//     PlcTask Inputs/GV_IO.diToolPresenceArmGripper2 <-> Channel 13/Input
//     PlcTask Inputs/GV_IO.diToolPresenceCone <-> Channel 8/Input
//   PLC_Tool_Magazine_8xx/PLC_Tool_Magazine_8xx Instance <-> Device 2 (EtherCAT)/U101.1 (EK1200)/IO273 (EL8601-8411)
//     PlcTask Inputs/GV_IO.aiToolPresenceRack <-> SlotGroup 4 (AI_1xV)/AI Inputs Channel 1/Value
//     PlcTask Inputs/GV_IO.biHandwheelCounterOverflow <-> SlotGroup 1 (CNT_2xDI)/ENC Inputs Channel 1/Status/Counter overflow
//     PlcTask Inputs/GV_IO.biHandwheelCounterUnderflow <-> SlotGroup 1 (CNT_2xDI)/ENC Inputs Channel 1/Status/Counter underflow
//     PlcTask Inputs/GV_IO.biHandwheelSetCounterDone <-> SlotGroup 1 (CNT_2xDI)/ENC Inputs Channel 1/Status/Set counter done
//     PlcTask Inputs/GV_IO.biSoftwareGateValid <-> SlotGroup 1 (CNT_2xDI)/ENC Inputs Channel 1/Status/Software gate valid
//     PlcTask Inputs/GV_IO.diHandwheelButtonFast <-> SlotGroup 2 (DI_4x)/DIP Inputs Channel 4/Input
//     PlcTask Inputs/GV_IO.diHandwheelButtonMinus <-> SlotGroup 1 (CNT_2xDI)/DIP Inputs Channel 2/Input
//     PlcTask Inputs/GV_IO.diHandwheelButtonPlus <-> SlotGroup 1 (CNT_2xDI)/DIP Inputs Channel 1/Input
//     PlcTask Inputs/GV_IO.diHandwheelIncrSelectorB0 <-> SlotGroup 2 (DI_4x)/DIP Inputs Channel 1/Input
//     PlcTask Inputs/GV_IO.diHandwheelIncrSelectorB1 <-> SlotGroup 2 (DI_4x)/DIP Inputs Channel 2/Input
//     PlcTask Inputs/GV_IO.diHandwheelIncrSelectorB2 <-> SlotGroup 2 (DI_4x)/DIP Inputs Channel 3/Input
//     PlcTask Inputs/GV_IO.diHandwheelTrackA <-> SlotGroup 1 (CNT_2xDI)/ENC Inputs Channel 1/Status/Status of input A
//     PlcTask Inputs/GV_IO.diHandwheelTrackB <-> SlotGroup 1 (CNT_2xDI)/ENC Inputs Channel 1/Status/Status of input B
//     PlcTask Inputs/GV_IO.udiHandwheelCounterValue <-> SlotGroup 1 (CNT_2xDI)/ENC Inputs Channel 1/Counter value
//     PlcTask Outputs/GV_IO.aoHandwheelPower <-> SlotGroup 5 (AO_1xV)/AO Outputs Channel 1/Analog output
//     PlcTask Outputs/GV_IO.boHandwheelSetCounter <-> SlotGroup 1 (CNT_2xDI)/ENC Outputs Channel 1/Control/Set counter
//     PlcTask Outputs/GV_IO.boSoftwareGateSet <-> SlotGroup 1 (CNT_2xDI)/ENC Outputs Channel 1/Control/Set software gate
//     PlcTask Outputs/GV_IO.doReserve27313 <-> SlotGroup 3 (PWM_OUT_DO)/DOS Outputs Channel 1/Output
//     PlcTask Outputs/GV_IO.pwmMagazineArmorFanOutput <-> SlotGroup 3 (PWM_OUT_DO)/PWM Outputs Channel 1/PWM output
//     PlcTask Outputs/GV_IO.pwmMagazineArmorFanPeriod <-> SlotGroup 3 (PWM_OUT_DO)/PWM Outputs Channel 1/PWM period
//     PlcTask Outputs/GV_IO.udoHandwheelCounterValue <-> SlotGroup 1 (CNT_2xDI)/ENC Outputs Channel 1/Set counter value
//   PLC_Tool_Magazine_8xx/PLC_Tool_Magazine_8xx Instance <-> Device 2 (EtherCAT)/U101.1 (EK1200)/O275 (EL2809)
//     PlcTask Outputs/GV_IO.doButtonUnlockMagazineDoorLamp <-> Channel 1/Output
//     PlcTask Outputs/GV_IO.doMagazineLight <-> Channel 9/Output
//     PlcTask Outputs/GV_IO.doReserve27510 <-> Channel 10/Output
//     PlcTask Outputs/GV_IO.doReserve27511 <-> Channel 11/Output
//     PlcTask Outputs/GV_IO.doReserve27512 <-> Channel 12/Output
//     PlcTask Outputs/GV_IO.doReserve27513 <-> Channel 13/Output
//     PlcTask Outputs/GV_IO.doReserve27514 <-> Channel 14/Output
//     PlcTask Outputs/GV_IO.doReserve27515 <-> Channel 15/Output
//     PlcTask Outputs/GV_IO.doReserve27516 <-> Channel 16/Output
//     PlcTask Outputs/GV_IO.doReserve2753 <-> Channel 3/Output
//     PlcTask Outputs/GV_IO.doReserve2754 <-> Channel 4/Output
//     PlcTask Outputs/GV_IO.doReserve2755 <-> Channel 5/Output
//     PlcTask Outputs/GV_IO.doReserve2757 <-> Channel 7/Output
//     PlcTask Outputs/GV_IO.doReserve2758 <-> Channel 8/Output
//     PlcTask Outputs/GV_IO.doSafetyAreaMagazineReset <-> Channel 6/Output
//     PlcTask Outputs/GV_IO.doUnlockMagazineDoor <-> Channel 2/Output
//   PLC_Tool_Magazine_8xx/PLC_Tool_Magazine_8xx Instance <-> NC-Task 1 SAF/Axes/A64.1 - Axis X
//     PlcTask Inputs/GV_Axes.stAxisX.stDriveAx8206.AxisRef.NcToPlc <-> Outputs/ToPlc
//     PlcTask Outputs/GV_Axes.stAxisX.stDriveAx8206.AxisRef.PlcToNc <-> Inputs/FromPlc
//   PLC_Tool_Magazine_8xx/PLC_Tool_Magazine_8xx Instance <-> NC-Task 1 SAF/Axes/A64.1 - Axis Z
//     PlcTask Inputs/GV_Axes.stAxisZ.stDriveAx8206.AxisRef.NcToPlc <-> Outputs/ToPlc
//     PlcTask Outputs/GV_Axes.stAxisZ.stDriveAx8206.AxisRef.PlcToNc <-> Inputs/FromPlc
//   PLC_Tool_Magazine_8xx/PLC_Tool_Magazine_8xx Instance <-> NC-Task 1 SAF/Axes/A64.2 - Axis Arm
//     PlcTask Inputs/GV_Axes.stAxisArm.stDriveAx8206.AxisRef.NcToPlc <-> Outputs/ToPlc
//     PlcTask Outputs/GV_Axes.stAxisArm.stDriveAx8206.AxisRef.PlcToNc <-> Inputs/FromPlc
//   PLC_Tool_Magazine_8xx/PLC_Tool_Magazine_8xx Instance <-> NC-Task 1 SAF/Axes/A64.2 - Axis Y
//     PlcTask Inputs/GV_Axes.stAxisY.stDriveAx8206.AxisRef.NcToPlc <-> Outputs/ToPlc
//     PlcTask Outputs/GV_Axes.stAxisY.stDriveAx8206.AxisRef.PlcToNc <-> Inputs/FromPlc
//   (this object) <-> Device 2 (EtherCAT)/U101.1 (EK1200)/A270.1/A64 (AX8620-0000-0105)/A64.1 (AX8206-0200-0107)
//     Drive/Inputs/In/nDataIn1 <-> Ch A/Ch A PositionControl Inputs/Ch A Following error actual value
//     Drive/Inputs/In/nDataIn3[0] <-> Ch A/Ch A TorqueControl Inputs/Ch A Torque/force actual value
//     Drive/Inputs/In/nDcOutputTime <-> InfoData/DcOutputShift
//     Drive/Inputs/In/nState1 <-> Ch A/Ch A AxisMain Inputs/Ch A Statusword
//     Drive/Inputs/In/nState2 <-> Ch A/Ch A AxisMain Inputs/Ch A Statusword @bit 8
//     Drive/Inputs/In/nState4 @bit 1 <-> WcState/InputToggle0
//     Drive/Inputs/In/nState4 <-> WcState/WcState0
//     Drive/Outputs/Out/nCtrl1 <-> Ch A/Ch A AxisMain Outputs/Ch A Controlword
//     Drive/Outputs/Out/nCtrl2 <-> Ch A/Ch A AxisMain Outputs/Ch A Controlword @bit 8
//     Drive/Outputs/Out/nDataOut1 <-> Ch A/Ch A Interpolator Outputs/Ch A Target position
//     Drive/Outputs/Out/nDataOut2 <-> Ch A/Ch A Interpolator Outputs/Ch A Target velocity
//     Enc/Inputs/In/nDataIn1 <-> Ch A/Ch A AxisMain Inputs/Ch A Position actual value
//     Enc/Inputs/In/nDcInputTime <-> InfoData/DcInputShift
//     Enc/Inputs/In/nState2 @bit 5 <-> Ch A/Ch A AxisMain Inputs/Position actual value invalid
//     Enc/Inputs/In/nState4 @bit 1 <-> WcState/InputToggle0
//     Enc/Inputs/In/nState4 <-> WcState/WcState0
//     Drive/Inputs/In/nDataIn1 <-> Ch B/Ch B PositionControl Inputs/Ch B Following error actual value
//     Drive/Inputs/In/nDataIn3[0] <-> Ch B/Ch B TorqueControl Inputs/Ch B Torque/force actual value
//     Drive/Inputs/In/nState1 <-> Ch B/Ch B AxisMain Inputs/Ch B Statusword
//     Drive/Inputs/In/nState2 <-> Ch B/Ch B AxisMain Inputs/Ch B Statusword @bit 8
//     Drive/Outputs/Out/nCtrl1 <-> Ch B/Ch B AxisMain Outputs/Ch B Controlword
//     Drive/Outputs/Out/nCtrl2 <-> Ch B/Ch B AxisMain Outputs/Ch B Controlword @bit 8
//     Drive/Outputs/Out/nDataOut1 <-> Ch B/Ch B Interpolator Outputs/Ch B Target position
//     Drive/Outputs/Out/nDataOut2 <-> Ch B/Ch B Interpolator Outputs/Ch B Target velocity
//     Enc/Inputs/In/nDataIn1 <-> Ch B/Ch B AxisMain Inputs/Ch B Position actual value
//     Enc/Inputs/In/nState2 @bit 5 <-> Ch B/Ch B AxisMain Inputs/Position actual value invalid
//   (this object) <-> Device 2 (EtherCAT)/U101.1 (EK1200)/A270.1/A64 (AX8620-0000-0105)/A64.2 (AX8206-0200-0107)
//     Drive/Inputs/In/nDataIn1 <-> Ch A/Ch A PositionControl Inputs/Ch A Following error actual value
//     Drive/Inputs/In/nDataIn3[0] <-> Ch A/Ch A TorqueControl Inputs/Ch A Torque/force actual value
//     Drive/Inputs/In/nDcOutputTime <-> InfoData/DcOutputShift
//     Drive/Inputs/In/nState1 <-> Ch A/Ch A AxisMain Inputs/Ch A Statusword
//     Drive/Inputs/In/nState2 <-> Ch A/Ch A AxisMain Inputs/Ch A Statusword @bit 8
//     Drive/Inputs/In/nState4 @bit 1 <-> WcState/InputToggle0
//     Drive/Inputs/In/nState4 <-> WcState/WcState0
//     Drive/Outputs/Out/nCtrl1 <-> Ch A/Ch A AxisMain Outputs/Ch A Controlword
//     Drive/Outputs/Out/nCtrl2 <-> Ch A/Ch A AxisMain Outputs/Ch A Controlword @bit 8
//     Drive/Outputs/Out/nDataOut1 <-> Ch A/Ch A Interpolator Outputs/Ch A Target position
//     Drive/Outputs/Out/nDataOut2 <-> Ch A/Ch A Interpolator Outputs/Ch A Target velocity
//     Enc/Inputs/In/nDataIn1 <-> Ch A/Ch A AxisMain Inputs/Ch A Position actual value
//     Enc/Inputs/In/nDcInputTime <-> InfoData/DcInputShift
//     Enc/Inputs/In/nState2 @bit 5 <-> Ch A/Ch A AxisMain Inputs/Position actual value invalid
//     Enc/Inputs/In/nState4 @bit 1 <-> WcState/InputToggle0
//     Enc/Inputs/In/nState4 <-> WcState/WcState0
//     Drive/Inputs/In/nDataIn1 <-> Ch B/Ch B PositionControl Inputs/Ch B Following error actual value
//     Drive/Inputs/In/nDataIn3[0] <-> Ch B/Ch B TorqueControl Inputs/Ch B Torque/force actual value
//     Drive/Inputs/In/nState1 <-> Ch B/Ch B AxisMain Inputs/Ch B Statusword
//     Drive/Inputs/In/nState2 <-> Ch B/Ch B AxisMain Inputs/Ch B Statusword @bit 8
//     Drive/Outputs/Out/nCtrl1 <-> Ch B/Ch B AxisMain Outputs/Ch B Controlword
//     Drive/Outputs/Out/nCtrl2 <-> Ch B/Ch B AxisMain Outputs/Ch B Controlword @bit 8
//     Drive/Outputs/Out/nDataOut1 <-> Ch B/Ch B Interpolator Outputs/Ch B Target position
//     Drive/Outputs/Out/nDataOut2 <-> Ch B/Ch B Interpolator Outputs/Ch B Target velocity
//     Enc/Inputs/In/nDataIn1 <-> Ch B/Ch B AxisMain Inputs/Ch B Position actual value
//     Enc/Inputs/In/nState2 @bit 5 <-> Ch B/Ch B AxisMain Inputs/Position actual value invalid

CONFIGURATION PLC_Tool_Magazine_8xx
    RESOURCE PLC ON TwinCAT3
        TASK PlcTask(INTERVAL := T#8ms, PRIORITY := 20);
        PROGRAM PRG_Main WITH PlcTask : PRG_Main;
    END_RESOURCE
END_CONFIGURATION

// ---- 02_Events/01_DUTs/02_ST/ST_Alarm.TcDUT
//-----------------------------------------------------------------------------------------
//
//                  				ST_Alarm
//
//								Variables alarme			
//-----------------------------------------------------------------------------------------
//
//Auteur: G.GOETZ (inspired by S.MANTZER)
//Création: 21.01.2026
//Dernière modification : 21.01.2026 (G.GOETZ)
//       			
//-----------------------------------------------------------------------------------------
//
//     							Liste des modifications  	
//
// 21.01.2026 (G.GOETZ) -> Création		
//-----------------------------------------------------------------------------------------

TYPE ST_Alarm :
STRUCT
	
	(** FB **)
	fbAlarm : FB_TcAlarm;

END_STRUCT
END_TYPE

// ---- 02_Events/01_DUTs/02_ST/ST_Event_Group.TcDUT
//-----------------------------------------------------------------------------------------
//
//                  				ST_Event_Group
//
//								Variables groupe d'évènements 			
//-----------------------------------------------------------------------------------------
//
//Auteur: G.GOETZ (inspired by S.MANTZER)
//Création: 21.01.2026
//Dernière modification : 21.01.2026 (G.GOETZ)
//       			
//-----------------------------------------------------------------------------------------
//
//     							Liste des modifications  	
//
// 21.01.2026 (G.GOETZ) -> Création		
//-----------------------------------------------------------------------------------------

TYPE ST_Event_Group :
STRUCT
	
	(** ARRAY ST **)
	aAlarm : ARRAY[1..GV_Events.iMaxAlarms] OF ST_Alarm ; // Alarms
	aMessage : ARRAY[1..GV_Events.iMaxMessages] OF ST_Message ; // Messages
	aOpMessage : ARRAY[1..GV_Events.iMaxOPMessages] OF ST_Alarm ; // Operator Messages
	
	(** FLAG **)
	bAlarmPresence : BOOL := FALSE ; // At last one alarm is present/activated
	
END_STRUCT
END_TYPE

// ---- 02_Events/01_DUTs/02_ST/ST_Message.TcDUT
//-----------------------------------------------------------------------------------------
//
//                  				ST_Message
//
//								Variables message			
//-----------------------------------------------------------------------------------------
//
//Auteur: G.GOETZ (inspired by S.MANTZER)
//Création: 21.01.2026
//Dernière modification : 21.01.2026 (G.GOETZ)
//       			
//-----------------------------------------------------------------------------------------
//
//     							Liste des modifications  	
//
// 21.01.2026 (G.GOETZ) -> Création		
//-----------------------------------------------------------------------------------------

TYPE ST_Message :
STRUCT
		
	(** FB **)
	fbMessage : FB_TcMessage;

END_STRUCT
END_TYPE

// ---- 03_Operating_Mode/01_DUTs/01_ENUM/ENUM_OpMode.TcDUT
{attribute 'qualified_only'}
{attribute 'strict'}

//-----------------------------------------------------------------------------------------
//
//                  				ENUM_OpMode
//
//								Enumération op Mode		
//-----------------------------------------------------------------------------------------
//
//Auteur: G.GOETZ
//Création: 20.02.2026
//Dernière modification : 20.02.2026 (G.GOETZ)
//       			
//-----------------------------------------------------------------------------------------
//
//     							Liste des modifications  	
//
// 20.02.2026 (G.GOETZ) -> Création		
//-----------------------------------------------------------------------------------------

TYPE ENUM_OpMode :
(
	None := 0 , // None mode
	AUTO := 1 , // AUTO mode
	MANU := 2 , // MANU mode
	INIT := 3 // INIT mode
);
END_TYPE

// ---- 05_Fans/01_DUTs/01_ENUM/ENUM_Fan_Type.TcDUT
{attribute 'qualified_only'}
{attribute 'strict'}

//-----------------------------------------------------------------------------------------
//
//                  				ENUM_Fan_Type
//
//						Enumération des types de ventilateur(s)			
//-----------------------------------------------------------------------------------------
//
//Auteur: G.GOETZ
//Création: 20.01.2026
//Dernière modification : 20.01.2026 (G.GOETZ)
//       			
//-----------------------------------------------------------------------------------------
//
//     							Liste des modifications  	
//
// 20.01.2026 (G.GOETZ) -> Création		
//-----------------------------------------------------------------------------------------

TYPE ENUM_Fan_Type :
(
	(*Unknow := 0 , // Unknow type*)
	PWM := 1 // With PWM type
);
END_TYPE

// ---- 05_Fans/01_DUTs/02_ST/ST_Fan.TcDUT
//-----------------------------------------------------------------------------------------
//
//                  				ST_Fan
//
//							Structure ventilateur(s) 			
//-----------------------------------------------------------------------------------------
//
//Auteur: G.GOETZ
//Création: 20.01.2026
//Dernière modification : 16.02.2026 (G.GOETZ)
//       			
//-----------------------------------------------------------------------------------------
//
//     							Liste des modifications  	
//
// 20.01.2026 (G.GOETZ) -> Création		
// 16.02.2026 (G.GOETZ) -> Ajout Sonde température PT-100
//-----------------------------------------------------------------------------------------

TYPE ST_Fan :
STRUCT
	
	(** SETUP ENUM **)
	eFanType : ENUM_Fan_Type ; // Type of the Fan

	(** SETUP REAL **)
	rTempStart : REAL := 30.0 ; // Temp in °C mini to start the Fan
	rTempMax : REAL := 45.0 ; // Temp in °C max speed of the Fan
	
	(** SETUP UINT **)
	uMinSpeed : UINT := 0 ; // Min Speed
	uMaxSpeed : UINT := 0 ; // Max Speed
	uMinPwm : UINT := 0 ; // Min Pwm at min speed (in %)
	uMaxPwm : UINT := 0 ; // Max Pwm at max speed (in %)
	uPwmPeriod : UINT := 0 ; // Period of the PWM signal (in ns)
	
	(** SETUP INT **)
	iEventGroup : INT := 0 ; // Group for events
	iIdHMI : INT := 0 ; // Number for events on HMI
	
	(** SETUP FLAG **)
	bEventAck : BOOL := FALSE ; // Events Acknowledgement
	bPresence : BOOL := FALSE ; // Fan presence or not

	(** PROCESS UINT **)
	uSpeedSet : UINT := 0 ; // Speed command (in tr/min)
	uPwmTarget : UINT := 0 ; // Taregt of the PWM signal, used to do a ramp
	uPwmOutput : UINT := 0 ; // Output of the PWM signal
	
	(** PROCESS INT **)

	(** PROCESS FLAG + R_TRIG **)
		bStart: BOOL := FALSE; // Start the Fan
			rtStart : R_TRIG ; // Trigger for Start the Fan
	
END_STRUCT
END_TYPE

// ---- 06_Doors/01_DUTs/01_ENUM/ENUM_Door_Type.TcDUT
{attribute 'qualified_only'}
{attribute 'strict'}

//-----------------------------------------------------------------------------------------
//
//                  				ENUM_Door_Type
//
//							Enumération des types de portes
//-----------------------------------------------------------------------------------------
//
//Auteur: G.GOETZ
//Création: 04.02.2026
//Dernière modification : 04.02.2026 (G.GOETZ)
//       			
//-----------------------------------------------------------------------------------------
//
//     							Liste des modifications  	
//
// 04.02.2026 (G.GOETZ) -> Création		
//-----------------------------------------------------------------------------------------

TYPE ENUM_Door_Type :
(
	Unknow := 0 ,
	AutoLockButtonUnlockOff := 1 ,
	AutoLockButtonUnlockOn := 2 
);
END_TYPE

// ---- 06_Doors/01_DUTs/02_ST/ST_Door.TcDUT
//-----------------------------------------------------------------------------------------
//
//                  				ST_Door
//
//								Structure porte(s) 			
//-----------------------------------------------------------------------------------------
//
//Auteur: G.GOETZ (inspired by S.MANTZER)
//Création: 13.01.2026
//Dernière modification : 13.01.2026 (G.GOETZ)
//       			
//-----------------------------------------------------------------------------------------
//
//     							Liste des modifications  	
//
// 13.01.2026 (G.GOETZ) -> Création		
//-----------------------------------------------------------------------------------------

TYPE ST_Door :
STRUCT

	(** SETUP ENUM **)
		eType : ENUM_Door_Type ; // Type of the Door
	
	(** SETUP INT **)
		iEventGroup : INT := 0 ; // Group for events
		iIdHMI : INT := 0 ; // Number for events on HMI
	
	(** SETUP FLAG **)
		bEventAck : BOOL := FALSE ; // Events Acknowledgement
		bPresence : BOOL := FALSE ; // Presence or not
	
	(** PROCESS INT **)

	(** PROCESS FLAG **)	
		bUnlockRequest : BOOL := FALSE ; // Request for unlock the door
		bUnlockRequestAck : BOOL := FALSE ; //Request for unlock the door acknowledgement
		bUnlockAuthorization : BOOL := FALSE ; // Authorization to unlock the door
		bLockRequest : BOOL := FALSE ; // Request for lock the door
		bLockRequestAck : BOOL := FALSE ; //Request for lock the door acknowledgement
		bLockAuthorization : BOOL := FALSE ; // Authorization to lock the door	
		
		bButtonUnlock : BOOL := FALSE ; // Button for unlock the door
		rtButtonUnlockTrig : R_trig ; // Trigger of the Button for unlock the door
		bButtonUnlockLamp : BOOL := FALSE ; // Lamp of the Button for unlock the door
		bButtonLock : BOOL := FALSE ; // Button for lock the door
		rtButtonLockTrig : R_trig ; // Trigger of the Button for lock the door
		bButtonLockLamp : BOOL := FALSE ; // Lamp of the Button for lock the door
		
		bUnlockOut : BOOL := FALSE ; // Output for unlock the door
		bLockOut : BOOL := FALSE ; // Output for lock the door
		
		bDoorOpen : BOOL := FALSE ; // Door is open
		bDoorCloseLock : BOOL := FALSE ; // Door is closed and locked
		bDoorSafetyRelay : BOOL := FALSE ; // Door safety relay
	
END_STRUCT
END_TYPE

// ---- 07_Cyltronic/01_DUTs/01_ENUM/ENUM_Cyltronic_Type.TcDUT
{attribute 'qualified_only'}
{attribute 'strict'}

//-----------------------------------------------------------------------------------------
//
//                  			ENUM_Cyltronic_Type
//
//							Enumération des types de Cyltronic
//-----------------------------------------------------------------------------------------
//
//Auteur: G.GOETZ
//Création: 04.03.2026
//Dernière modification : 04.03.2026 (G.GOETZ)
//       			
//-----------------------------------------------------------------------------------------
//
//     							Liste des modifications  	
//
// 04.03.2026 (G.GOETZ) -> Création		
//-----------------------------------------------------------------------------------------

TYPE ENUM_Cyltronic_Type :
(
	Unknow := 0 ,
	IOLink := 1 ,
	DiDo := 2 
);
END_TYPE

// ---- 07_Cyltronic/01_DUTs/01_ENUM/teCTCBrakeMode.TcTLEO
TYPE teCTCBrakeMode :
(
	CTC_BRAKE_MODE_OFF := 0,
	CTC_BRAKE_MODE_WHEN_DISABLED := 1,
	CTC_BRAKE_MODE_IN_STANDSTILL := 2
);
END_TYPE

// ---- 07_Cyltronic/01_DUTs/01_ENUM/teCTCConfigStep.TcDUT
TYPE teCTCConfigStep :
(
	CTC_CONFIG_IDLE,
	CTC_CONFIG_READ_START,
	CTC_CONFIG_READ_WAIT,
	CTC_CONFIG_READ_FINISH,
	CTC_CONFIG_WRITE_PREPARE,
	CTC_CONFIG_WRITE_START,
	CTC_CONFIG_WRITE_WAIT
);
END_TYPE

// ---- 07_Cyltronic/01_DUTs/01_ENUM/teCTCDeviceStatus.TcTLEO
TYPE teCTCDeviceStatus :
(
	DEVICE_OK 				:= 0,
	MAINTENANCE_REQUIRED 	:= 1,
	OUT_OF_SPECIFICATION 	:= 2,
	FUNCTIONAL_CHECK 		:= 3,
	FAILURE 				:= 4
);
END_TYPE

// ---- 07_Cyltronic/01_DUTs/01_ENUM/teCTCEvent.TcTLEO
TYPE teCTCEvent :
(
	CTC_NO_EVENT 					:= 0,
	CTC_EVENT_UNDERTEMP_MC 			:= 6210,
	CTC_EVENT_OVERTEMP_MC 			:= 6211,
	CTC_EVENT_UNDERTEMP_CB 			:= 6212,
	CTC_EVENT_OVERTEMP_CB 			:= 6213,
	CTC_EVENT_UNDERTEMP_EB 			:= 6214,
	CTC_EVENT_OVERTEMP_EB 			:= 6215,
	CTC_EVENT_OVERTEMP_PS_PHASE_U 	:= 6216,
	CTC_EVENT_OVERTEMP_PS_PHASE_V 	:= 6217,
	CTC_EVENT_OVERTEMP_PS_PHASE_W 	:= 6218,
	CTC_EVENT_OVERTEMP_MOT_PHASE_U 	:= 6219,
	CTC_EVENT_OVERTEMP_MOT_PHASE_V 	:= 6220,
	CTC_EVENT_OVERTEMP_MOT_PHASE_W 	:= 6221,
	CTC_EVENT_CONTROLLER_ERROR 		:= 6222,
	CTC_EVENT_INTERNAL_ERROR 		:= 6223,
	CTC_EVENT_TRACKING_ERROR 		:= 6224,
	CTC_EVENT_INVALID_SETPOINTS 	:= 6225,
	CTC_EVENT_OVERVOLTAGE_LOGIC 	:= 20752,
	CTC_EVENT_UNDERVOLTAGE_LOGIC 	:= 20753,
	CTC_EVENT_OVERVOLTAGE_POWER 	:= 20754,
	CTC_EVENT_HOMING_FAILED 		:= 6226
);
END_TYPE

// ---- 07_Cyltronic/01_DUTs/01_ENUM/teCTCGDSStep.TcDUT
TYPE teCTCGDSStep :
(
	CTC_GDS_IDLE,
	CTC_GDS_READ_STATUS_START,
	CTC_GDS_READ_STATUS_WAIT,
	CTC_GDS_READ_DETSTAT_START,
	CTC_GDS_READ_DETSTAT_WAIT
);
END_TYPE

// ---- 07_Cyltronic/01_DUTs/01_ENUM/teCTCHomeMode.TcTLEO
TYPE teCTCHomeMode :
(
	CTC_HOME_MODE_DIRECT 		:= 0,
	CTC_HOME_MODE_ENDSTOPIN 	:= 1,
	CTC_HOME_MODE_ENDSTOPOUT 	:= 2
);
END_TYPE

// ---- 07_Cyltronic/01_DUTs/01_ENUM/teCTCStep.TcTLEO
TYPE teCTCStep :
(
	FB_CTC_FUNCTIONBLOCK_DISABLED 	:= 0,
	FB_CTC_CONNECTING 				:= 1,
	FB_CTC_DISABLED 				:= 2,
	FB_CTC_ENABLING					:= 21,
	FB_CTC_DISABLING				:= 22,
	FB_CTC_HOME 					:= 3,
	FB_CTC_TEACH 					:= 4,
	FB_CTC_READY 					:= 5,
	FB_CTC_MOVE_OUT 				:= 6,
	FB_CTC_MOVE_IN 					:= 7,
	FB_CTC_MOVE_ABSOLUTE 			:= 8,	
	FB_CTC_MOVE_CONTINUOUS 			:= 9,
	FB_CTC_HALTING 					:= 10,
	FB_CTC_ERROR 					:= 11,
	FB_CTC_RESET 					:= 12
);
END_TYPE

// ---- 07_Cyltronic/01_DUTs/01_ENUM/teCTCWarningID.TcTLEO
TYPE teCTCWarningID :
(
	CTC_WARNING_OK 				:= 0,
	CTC_WARNING_FB_SETPOINTS 	:= 1,
	CTC_WARNING_FB_COMMAND 		:= 2,
	CTC_WARNING_EVENT 			:= 3
);
END_TYPE

// ---- 07_Cyltronic/01_DUTs/02_ST/ST_Cyltronic.TcDUT
//-----------------------------------------------------------------------------------------
//
//                  				ST_Cyltronic
//
//								Structure Cyltronic
//-----------------------------------------------------------------------------------------
//
//Auteur: G.GOETZ
//Création: 04.03.2026
//Dernière modification : 04.03.2026 (G.GOETZ)
//       			
//-----------------------------------------------------------------------------------------
//
//     							Liste des modifications  	
//
// 04.03.2026 (G.GOETZ) -> Création		
//-----------------------------------------------------------------------------------------

TYPE ST_Cyltronic :
STRUCT

	(** SETUP T_AmsNetID **)
		(* For IO/Link *)
			netID : T_AmsNetID ;

	(** SETUP ENUM **)
		eType : ENUM_Cyltronic_Type ; // Type
		(* For IO/Link *)
			ePort : E_IolPort ; // Port on the EL6224
			eState : teCTCStep ; // State
				
	(** SETUP INT **)
		iEventGroup : INT := 0 ; // Group for events
		iIdHMI : INT := 0 ; // Number for events on HMI
	
	(** SETUP FLAG **)
		bEventAck : BOOL := FALSE ; // Events Acknowledgement
		bPresence : BOOL := FALSE ; // Presence or not
	
	(** ALARMS FLAG **)
		bAlDriveFault : BOOL := FALSE ; // Drive in Fault
	
	(** PROCESS ARRAY **)
		(* For IO/Link *)
			aProcessDataInRaw AT %I* : ARRAY[0..13] OF BYTE ;
			aProcessDataOutRaw AT %Q* : ARRAY[0..7] OF BYTE ; 
	
	(** PROCESS REAL **)
		(* For IO/Link *)
			(*Jog*)
				lrJogPos : REAL ; // Jog Position
				lrJogVel : REAL ; // Jog Velocity
				lrJogAccDec : LREAL ; // Jog Acceleration and Deceleration
				lrJogForce : LREAL ; // Jog Force
			(*Auto*)
				lrAutoPos : LREAL ; // AUTO Postion
				lrAutoVel : LREAL ; // AUTO Velocity
				lrAutoAccDec : LREAL ; // AUTO Acceleration
				lrAutoForce : LREAL ; // Jog Force
	
	(** PROCESS INT **)

	(** PROCESS FLAG + R_TRIG **)
		(* For IO/Link *)
			(*Power*)
				bPowerEnable : BOOL := FALSE ; // Can be Powered
			(*Halt*)
				bHaltExecute : BOOL := FALSE ; // Execute a STOP
				bHaltDone : BOOL := FALSE ; // STOP is Done
		bAuthorizationManuCyltronicRest : BOOL ; // Authorization to move to Rest in Manual
		bAuthorizationManuCyltronicWork : BOOL ; // Authorization to move to Work in Manual
		bAuthorizationAutoCyltronicRest : BOOL ; // Authorization to move to Rest in AUTO
		bAuthorizationAutoCyltronicWork : BOOL ; // Authorization to move to Work in AUTO
		
		bReleaseBreakOutput AT %Q* : BOOL ;

		bWorkPositionCmd : BOOL := FALSE ; // Command to go to work position
			rtWorkPositionCmd : R_TRIG ; // Trigger of the command to go to work position
		bWorkPositionDone : BOOL := FALSE ; // Go to work position is Done
		bRestPositionCmd : BOOL := FALSE ; // Command to go to rest position
			rtRestPositionCmd : R_TRIG ; // Trigger of the command to go to rest position
		bRestPositionDone : BOOL := FALSE ; // Go to rest position is Done
	
		(* For IO/Link *)
			bStartWriteConfig : BOOL := FALSE ; // Start for write the config
	
	(** PROCESS ST **)
		(* For IO/Link *)
			stProcessDataIn : tstCTCProcessDataIn ; // Process Data In
			stProcessDataOut : tstCTCProcessDataOut ; // Process Data Out
		
			stConfigDefault : tstCTCConfiguration ; // Default Configuration
			stConfigRead : tstCTCConfiguration ; // Configuration Read
			stConfigWrite : tstCTCConfiguration ; // Configuration Write
			stParameters : tstCTCParameters ; // Parameters
			
			stStatus : tstCTCDeviceStatus ; // Status
		
END_STRUCT
END_TYPE

// ---- 07_Cyltronic/01_DUTs/02_ST/tstCTCConfiguration.TcDUT
TYPE tstCTCConfiguration :
STRUCT
	MaxSpeedFreePositioning	:REAL := 600.0;	
	MaxForceFreePositioning	:REAL := 400.0;	
	MaxAccDec				:REAL := 5.0;	
	EndPositionIn			:REAL := 0.0;	
	EndPositionOut			:REAL := 100.0;	
	HomeMode				:teCTCHomeMode := CTC_HOME_MODE_ENDSTOPIN;
END_STRUCT
END_TYPE

// ---- 07_Cyltronic/01_DUTs/02_ST/tstCTCConfigVariable.TcDUT
TYPE tstCTCConfigVariable :
STRUCT
	Name 			:STRING[64];
	Index 			:WORD;
	Subindex 		:BYTE;
	DataType 		:USINT := 0; 	// 0=Real, 1=Usint
	ValueIfReal 	:REAL;
	ValueIfUSINT 	:USINT;
END_STRUCT
END_TYPE

// ---- 07_Cyltronic/01_DUTs/02_ST/tstCTCDeviceStatus.TcDUT
TYPE tstCTCDeviceStatus :
STRUCT
	DeviceStatus 	:teCTCDeviceStatus; 			// Index 36: Device Status
	Events 			:ARRAY[0..4]OF tstCTCEvent; 	// Index 37: First 5 pending Events
END_STRUCT
END_TYPE

// ---- 07_Cyltronic/01_DUTs/02_ST/tstCTCEvent.TcDUT
TYPE tstCTCEvent :
STRUCT
	Qualifier 	:USINT; 		// 1 byte event qualifier
	Event 		:teCTCEvent; 	// 2 byte event, converted to enum type
END_STRUCT
END_TYPE

// ---- 07_Cyltronic/01_DUTs/02_ST/tstCTCInternalCommands.TcDUT
TYPE tstCTCInternalCommands :
STRUCT
	bHome 			:BOOL;
	bTeach 			:BOOL;
	bMoveAbsolute 	:BOOL;
	bHalt 			:BOOL;
	bMoveIn 		:BOOL;
	bMoveOut 		:BOOL;
	bMoveContinuous :BOOL;
END_STRUCT
END_TYPE

// ---- 07_Cyltronic/01_DUTs/02_ST/tstCTCParameters.TcDUT
TYPE tstCTCParameters :
STRUCT
	TargetPosition		:REAL := 0.0;		// [mm]
	TargetVelocity		:REAL := 600.0;		// [mm/s]
	TargetAccDec		:REAL := 5.0;		// [m/s^2]
	TargetForce			:REAL := 400.0;		// [N]
END_STRUCT
END_TYPE

// ---- 07_Cyltronic/01_DUTs/02_ST/tstCTCProcessDataIn.TcDUT
TYPE tstCTCProcessDataIn :
STRUCT
	State			:USINT;		
	stStatusBits	:tstCTCStatusBits;	
	ActualForce 	:REAL;		
	ActualSpeed 	:REAL;		
	ActualPosition 	:REAL;		
END_STRUCT
END_TYPE

// ---- 07_Cyltronic/01_DUTs/02_ST/tstCTCProcessDataOut.TcDUT
TYPE tstCTCProcessDataOut :
STRUCT
	MotionMode		:USINT;	
	TargetPosition	:REAL;	
	Override1		:USINT; 
	Override2		:USINT; 
	Override3		:USINT; 	
END_STRUCT
END_TYPE

// ---- 07_Cyltronic/01_DUTs/02_ST/tstCTCStatusBits.TcDUT
TYPE tstCTCStatusBits :
STRUCT
	TrackingErrorToleranceExceeded 	:BOOL;
	WarningActive					:BOOL;
	MotionModeActive				:BOOL;
	MotionCommandCompleted 			:BOOL;	
	LimitSwitchIn					:BOOL;	
	LimitSwitchOut					:BOOL;
	Homed							:BOOL;
	Ready							:BOOL;
END_STRUCT
END_TYPE

// ---- 07_Cyltronic/01_DUTs/03_Union/tuReal.TcDUT
TYPE tuReal:
UNION
	rReal	:REAL;
	aBytes	:ARRAY[0..3] OF BYTE;
END_UNION
END_TYPE

// ---- 08_Cycle/01_DUTs/01_ENUM/ENUM_Cycle_Action.TcDUT
{attribute 'qualified_only'}
{attribute 'strict'}

//-----------------------------------------------------------------------------------------
//
//                  				ENUM_Cycle_Action
//
//							Enumération des actions du cycle			
//-----------------------------------------------------------------------------------------
//
//Auteur: G.GOETZ
//Création: 04.02.2026
//Dernière modification : 04.02.2026 (G.GOETZ)
//       			
//-----------------------------------------------------------------------------------------
//
//     							Liste des modifications  	
//
// 04.02.2026 (G.GOETZ) -> Création		
//-----------------------------------------------------------------------------------------

TYPE ENUM_Cycle_Action :
(
    None := 0 , // No action
    PickToolMagazine := 1 , // Pick tool in magazine with the manipulator head
    ManipulatorToArm := 2 , // Transfer tool from the manipulator head to the changing arm
    ArmCNC := 3 , // Transfer between changing arm and CNC
    ArmToManipulator := 4 , // Transfer tool from the changing arm to the manipulator head
    PlaceToolMagazine := 5 , // Place tool in magazine with the manipulator head
	
	HomePosition := 200 , 
	
	PickPlaceToolMag1 := 211 ,
	PickPlaceToolMag2 := 212 ,
	PickPlaceToolMag3 := 213 ,
	PickPlaceToolMag4 := 214 ,
	PickPlaceToolMag5 := 215
);
END_TYPE

// ---- 08_Cycle/01_DUTs/01_ENUM/ENUM_Cycle_Step.TcDUT
{attribute 'qualified_only'}
{attribute 'strict'}

//-----------------------------------------------------------------------------------------
//
//                  				ENUM_Cycle_Step
//
//							Enumération des étapes du cycle			
//-----------------------------------------------------------------------------------------
//
//Auteur: G.GOETZ
//Création: 02.02.2026
//Dernière modification : 02.02.2026 (G.GOETZ)
//       			
//-----------------------------------------------------------------------------------------
//
//     							Liste des modifications  	
//
// 02.02.2026 (G.GOETZ) -> Création		
//-----------------------------------------------------------------------------------------

TYPE ENUM_Cycle_Step :
(
	InitAll := 0 , // Init All
	InitData := 1 , // Init Data
	Ready := 2 , // Ready
	Preparation := 3 , // Tool Preparation/Anticipation
	BuildSequence := 4 , // Build the Sequence
	ExecuteSequence := 5 , // Execute the Sequence
	End := 7 , // End
	Abort := 8 , // Abort
	Error := 9 // Error
);
END_TYPE

// ---- 08_Cycle/01_DUTs/01_ENUM/ENUM_Cycle_Type.TcDUT
{attribute 'qualified_only'}
{attribute 'strict'}

//-----------------------------------------------------------------------------------------
//
//                  				ENUM_Cycle_Type
//
//							Enumération des types de cycle			
//-----------------------------------------------------------------------------------------
//
//Auteur: G.GOETZ
//Création: 24.02.2026
//Dernière modification : 24.02.2026 (G.GOETZ)
//       			
//-----------------------------------------------------------------------------------------
//
//     							Liste des modifications  	
//
// 24.02.2026 (G.GOETZ) -> Création		
//-----------------------------------------------------------------------------------------

TYPE ENUM_Cycle_Type :
(
	None := 0 , // None
	LoadSmallBig := 1 , // Load only : small or big tool (A100=small / A200=big)
	UnloadSmall := 2 , // Unload only : small tool (B100=small)
	UnloadBig := 3 , // Unload only : big tool (B200=big)
	LoadSmallUnloadSmall := 4 , // Load : small tool / Unload : small tool (C100=small/small)
	
	//LoadBigUnloadBig := 5 , // Load : big tool / Unload : big tool (D100=big/big)
	//LoadBigUnloadSmall := 6 , // Load : big tool / Unload : small tool (D200=big/small)
	//LoadSmallUnloadBig := 7 , // Load : small tool / Unload : big tool (D300=small/big)

	// Dxxx = Cycle in two step -> "UnloadSmall/Big" and after "LoadSmallBig"

	EssaiType1 := 101 , // EsaiType1

	Essai_1 := 201 ,
	Essai_1_2 := 202 ,
	Essai_1_3 := 203 
	
);
END_TYPE

// ---- 09_Tool_Magazine/01_DUTs/01_ENUM/ENUM_Gripper_Mode.TcDUT
{attribute 'qualified_only'}
{attribute 'strict'}

//-----------------------------------------------------------------------------------------
//
//                  			ENUM_Gripper_Mode
//
//			Enumération des modes de mouvements de la pince du manipulateur			
//-----------------------------------------------------------------------------------------
//
//Auteur: G.GOETZ
//Création: 05.02.2026
//Dernière modification : 05.02.2026 (G.GOETZ)
//       			
//-----------------------------------------------------------------------------------------
//
//     							Liste des modifications  	
//
// 05.02.2026 (G.GOETZ) -> Création		
//-----------------------------------------------------------------------------------------

TYPE ENUM_Gripper_Mode :
(
	Open := 0 , // Open the gripper
	Close := 1 // CLose the gripper
);
END_TYPE

// ---- 09_Tool_Magazine/01_DUTs/01_ENUM/ENUM_Position_Axis.TcDUT
{attribute 'qualified_only'}
{attribute 'strict'}

//-----------------------------------------------------------------------------------------
//
//                  				ENUM_Door
//
//						Enumération des types de porte(s)			
//-----------------------------------------------------------------------------------------
//
//Auteur: G.GOETZ
//Création: 13.01.2026
//Dernière modification : 13.01.2026 (G.GOETZ)
//       			
//-----------------------------------------------------------------------------------------
//
//     							Liste des modifications  	
//
// 13.01.2026 (G.GOETZ) -> Création		
//-----------------------------------------------------------------------------------------

TYPE ENUM_Position_Axis :
(
	Unknow := 0 , // Unknow position
	Work1 := 10 , // At Work position
	Work2 := 20 , // At Work position
	Work3 := 30 , // At Work position
	Work4 := 40 , // At Work position
	Work5 := 50 , // At Work position

	CNC := 80 , // At CNC position
	Ref := 90 , // At Ref position
	Home := 100 // At Home position
);
END_TYPE

// ---- 09_Tool_Magazine/01_DUTs/01_ENUM/ENUM_Position_Magazine.TcDUT
{attribute 'qualified_only'}
{attribute 'strict'}

//-----------------------------------------------------------------------------------------
//
//                  				ENUM_Door
//
//						Enumération des types de porte(s)			
//-----------------------------------------------------------------------------------------
//
//Auteur: G.GOETZ
//Création: 13.01.2026
//Dernière modification : 13.01.2026 (G.GOETZ)
//       			
//-----------------------------------------------------------------------------------------
//
//     							Liste des modifications  	
//
// 13.01.2026 (G.GOETZ) -> Création		
//-----------------------------------------------------------------------------------------

TYPE ENUM_Position_Magazine :
(
	Unknow := 0 , // Unknow position
	Top := 1 , // At the top of the Magazine
	Bottom := 2 // At the bootom of the Magazine 
);
END_TYPE

// ---- 09_Tool_Magazine/01_DUTs/01_ENUM/ENUM_Tool_Type.TcDUT
{attribute 'qualified_only'}
{attribute 'strict'}

//-----------------------------------------------------------------------------------------
//
//                  				ENUM_Tool_Type
//
//							Enumération des types d'outils			
//-----------------------------------------------------------------------------------------
//
//Auteur: G.GOETZ
//Création: 14.01.2026
//Dernière modification : 14.01.2026 (G.GOETZ)
//       			
//-----------------------------------------------------------------------------------------
//
//     							Liste des modifications  	
//
// 14.01.2026 (G.GOETZ) -> Création		
//-----------------------------------------------------------------------------------------

TYPE ENUM_Tool_Type :
(
	Unknow := 0 , // Unknow type
	Small := 1 , // Small tool
	Big := 2 , // Big tool
	GPS70 := 3 // GPS70 
);
END_TYPE

// ---- 09_Tool_Magazine/01_DUTs/01_ENUM/ENUM_Tunnel_Mode.TcDUT
{attribute 'qualified_only'}
{attribute 'strict'}

//-----------------------------------------------------------------------------------------
//
//                  			ENUM_Tunnel_Mode
//
//			Enumération des modes de passage du tunnel par le manipulateur			
//-----------------------------------------------------------------------------------------
//
//Auteur: G.GOETZ
//Création: 06.02.2026
//Dernière modification : 06.02.2026 (G.GOETZ)
//       			
//-----------------------------------------------------------------------------------------
//
//     							Liste des modifications  	
//
// 06.02.2026 (G.GOETZ) -> Création		
//-----------------------------------------------------------------------------------------

TYPE ENUM_Tunnel_Mode :
(
	TopToBottom := 0 , // Tunnel way : Top -> Bottom
	BottomToTop := 1 // Tunnel way : Bottom -> Top
);
END_TYPE

// ---- 09_Tool_Magazine/01_DUTs/02_ST/ST_Changing_Arm.TcDUT
//-----------------------------------------------------------------------------------------
//
//                  				ST_Changing_Arm
//
//								Structure bras changeur		
//-----------------------------------------------------------------------------------------
//
//Auteur: G.GOETZ
//Création: 03.02.2026
//Dernière modification : 03.02.2026 (G.GOETZ)
//       			
//-----------------------------------------------------------------------------------------
//
//     							Liste des modifications  	
//
// 03.02.2026 (G.GOETZ) -> Création		
//-----------------------------------------------------------------------------------------

TYPE ST_Changing_Arm :
STRUCT
	
	(** ARRAY ST **)
		aGripper : ARRAY[1..2] OF ST_Changing_Arm_Gripper ; // Changing_Arm_Gripper structure
	
	(** ALARMS FLAG **)
		bAlAlarme1 : BOOL ; // Alarme 1 alarm

	(** SETUP FLAG **)
		bAck : BOOL :=FALSE; // Event acknowledgement
		
	(** PROCESS ENUM **)
		ePositionAxis : ENUM_Position_Axis ; // Position of the Changing Arm
	
	(** PROCESS LREAL **)
		lrArmPosition : LREAL ; // Arm position
		lrArmPositionTol : LREAL ; // Arm Position Tolerance
		
		lrArmHome : LREAL ; // Arm coordinate at Home
		lrArmManipulator : LREAL ; // Arm coordinate at transfer position (Arm<->Manipuator)
		lrArmCnc: LREAL ; // Arm coordinate at transfer position (Arm<->Cnc)
	
END_STRUCT
END_TYPE

// ---- 09_Tool_Magazine/01_DUTs/02_ST/ST_Changing_Arm_Gripper.TcDUT
TYPE ST_Changing_Arm_Gripper :
STRUCT
	
	(** ST **)
		stLocationMemory : ST_Tool_Location ; // Tool_Location structure
	
	(** PROCESS INT **)
		iAbsLocationNumberMemory : INT := 0 ; // Memory -> Number of the location in the Magazine
		iRelLocationNumberMemory : INT ; // Memory -> Number of the location in relative in the Magazine
		
	(** PROCESS FLAG **)
		bToolPresenceMemory : BOOL ; // Memory -> Tool Presence in the Manipulator
	
END_STRUCT
END_TYPE

// ---- 09_Tool_Magazine/01_DUTs/02_ST/ST_Manipulator_Head.TcDUT
//-----------------------------------------------------------------------------------------
//
//                  				ST_Manipulator_Head
//
//								Structure tête manipulateur			
//-----------------------------------------------------------------------------------------
//
//Auteur: G.GOETZ
//Création: 27.01.2026
//Dernière modification : 27.01.2026 (G.GOETZ)
//       			
//-----------------------------------------------------------------------------------------
//
//     							Liste des modifications  	
//
// 27.01.2026 (G.GOETZ) -> Création		
//-----------------------------------------------------------------------------------------

TYPE ST_Manipulator_Head :
STRUCT	

	(** ALARMS FLAG **)
		bAlAlarme1 : BOOL ; // Alarme 1 alarm
	
	(** SETUP FLAG **)
		bAck : BOOL := FALSE ; // Event acknowledgement
	
	(** PROCESS ENUM **)
		ePositionMag : ENUM_Position_Magazine ; // Position of the Manipulator Head in the magazine
		ePositionHome : ENUM_Position_Magazine ; // Position of the Home in the magazine
		
		ePositionAxis : ENUM_Position_Axis ; // Position of the Manipulator Head
	
	(** PROCESS LREAL **)
		lrXPosition : LREAL ; // X Position of the manipulator
		lrYPosition : LREAL ; // Y Position of the manipulator
		lrZPosition : LREAL ; // Z Position of the manipulator
		lrXPositionTol : LREAL ; // X Position Tolerance
		lrYPositionTol : LREAL ; // Y Position Tolerance
		lrZPositionTol : LREAL ; // Z Position Tolerance
		
		lrXHome : LREAL ; // X coordinate at Home
		lrYHome : LREAL ; // Y coordinate at Home
		lrZHome : LREAL ; // Z coordinate at Home
		
		lrXTunnel : LREAL ; // X coordinate at Tunnel
		lrYTunnel : LREAL ; // Y coordinate at Tunnel
		lrZTunnelTop : LREAL ; // Z coordinate at Tunnel (Top)
		lrZTunnelBottom : LREAL ; // Z coordinate at Tunnel (Bottom)
		
		lrXBreakage : LREAL ; // X coordinate at breakage sensor
		lrYBreakage : LREAL ; // Y coordinate at breakage sensor
		lrZBreakage : LREAL ; // Z coordinate at breakage sensor
		
		//lrXReadyTransfer : LREAL ; // X coordinate to be ready for the transfer to the Changing Arm
		//lrYReadyTransfer : LREAL ; // Y coordinate to be ready for the transfer to the Changing Arm
		//lrZReadyTransfer : LREAL ; // Z coordinate to be ready for the transfer to the Changing Arm
		
		lrXTransferGripper1 : LREAL ; // X coordinate at transfer to the Changing Arm gripper 1
		lrYTransferGripper1 : LREAL ; // Y coordinate at transfer to the Changing Arm gripper 1
		lrZTransferGripper1 : LREAL ; // Z coordinate at transfer to the Changing Arm gripper 1

		lrXTransferGripper2 : LREAL ; // X coordinate at transfer to the Changing Arm gripper 2
		lrYTransferGripper2 : LREAL ; // Y coordinate at transfer to the Changing Arm gripper 2
		lrZTransferGripper2 : LREAL ; // Z coordinate at transfer to the Changing Arm gripper 2
	
	(** PROCESS FLAG **)
		bAuthorizationManuGripperClose : BOOL ; // Authorization to close the Manipulator Gripper in Manual
		bAuthorizationManuGripperOpen : BOOL ; // Authorization to open the Mnipulator Gripper in Manual
		
		bCtrlBreakage : BOOL ; // Breakage ctrl in progress, for velocity
		
	(** ST **)
		stLocationMemory : ST_Tool_Location ; // Tool_Location structure
	
	(** PROCESS INT **)
		iAbsLocationNumberMemory : INT := 0 ; // Memory -> Number of the location in the Magazine
		iRelLocationNumberMemory : INT ; // Memory -> Number of the location in relative in the Magazine
		
	(** PROCESS FLAG **)
		bToolPresenceMemory : BOOL ; // Memory -> Tool Presence in the Manipulator
		
		bInterferingArm : BOOL ; // Manipulator is interfering with the Changing Arm

END_STRUCT
END_TYPE

// ---- 09_Tool_Magazine/01_DUTs/02_ST/ST_Tool_Corrector_M.TcDUT
//-----------------------------------------------------------------------------------------
//
//                  				ST_Tool_Corrector_M
//
//								Structure correcteur M outil 			
//-----------------------------------------------------------------------------------------
//
//Auteur: G.GOETZ (inspired by S.FLEURY)
//Création: 20.01.2026
//Dernière modification : 20.01.2026 (G.GOETZ)
//       			
//-----------------------------------------------------------------------------------------
//
//     							Liste des modifications  	
//
// 20.01.2026 (G.GOETZ) -> Création		
//-----------------------------------------------------------------------------------------

TYPE ST_Tool_Corrector_M :
STRUCT
	
	(** SETUP DINT **)
		Longueur : DINT ;
		UsureLongueur : DINT ;
		Rayon : DINT ;
		UsureRayon : DINT ;
		PositionW : DINT ;
		
END_STRUCT
END_TYPE

// ---- 09_Tool_Magazine/01_DUTs/02_ST/ST_Tool_Corrector_T.TcDUT
//-----------------------------------------------------------------------------------------
//
//                  				ST_Tool_Corrector_T
//
//								Structure correcteur T outil 			
//-----------------------------------------------------------------------------------------
//
//Auteur: G.GOETZ (inspired by S.FLEURY)
//Création: 20.01.2026
//Dernière modification : 20.01.2026 (G.GOETZ)
//       			
//-----------------------------------------------------------------------------------------
//
//     							Liste des modifications  	
//
// 20.01.2026 (G.GOETZ) -> Création		
//-----------------------------------------------------------------------------------------

TYPE ST_Tool_Corrector_T :
STRUCT
	
	(** SETUP DINT **)
		Longueur : DINT ;
		UsureLongueur : DINT ;
		Rayon : DINT ;
		PositionW : DINT ;
		LongY : DINT ;
		UsureY : DINT ;
		LontZ : DINT ;
		UsureZ : DINT ;
		Quadrant : DINT ;
	
END_STRUCT
END_TYPE

// ---- 09_Tool_Magazine/01_DUTs/02_ST/ST_Tool_Name.TcDUT
//-----------------------------------------------------------------------------------------
//
//                  				ST_Tool_Name
//
//								Structure nom outil 			
//-----------------------------------------------------------------------------------------
//
//Auteur: G.GOETZ (inspired by S.FLEURY)
//Création: 20.01.2026
//Dernière modification : 20.01.2026 (G.GOETZ)
//       			
//-----------------------------------------------------------------------------------------
//
//     							Liste des modifications  	
//
// 20.01.2026 (G.GOETZ) -> Création		
//-----------------------------------------------------------------------------------------

TYPE ST_Tool_Name :
STRUCT
	
	(** SETUP STRING **)
		Name : STRING[GV_Tool_Magazine.iNumCharaToolName] ; // Name
	
END_STRUCT
END_TYPE

// ---- 09_Tool_Magazine/01_DUTs/02_ST/ST_Tool_Parameters.TcDUT
//-----------------------------------------------------------------------------------------
//
//                  				ST_Tool_Parameters
//
//								Structure paramètres outil 			
//-----------------------------------------------------------------------------------------
//
//Auteur: G.GOETZ (inspired by S.FLEURY)
//Création: 14.01.2026
//Dernière modification : 14.01.2026 (G.GOETZ)
//       			
//-----------------------------------------------------------------------------------------
//
//     							Liste des modifications  	
//
// 14.01.2026 (G.GOETZ) -> Création		
//-----------------------------------------------------------------------------------------

TYPE ST_Tool_Parameters : // The order of the structure is important
STRUCT

	Number : DINT ; // Tool Number = Numéro outil
	LifetimeInit : DINT ; // Initial Lifetime of the Tool = Durée de vie initiale
	LifetimeRemain : DINT ; // Remaining Lifetime = Durée de vie restante
    Location : UINT ; // Location of the Tool in the Magazine = Emplacement godet dans magasin
    TwinNumber : BYTE ; // Number of the twin Tool = Numéro outil jumeaux
    Size : BYTE ; // Tool Size = Taille outil
    State :  BYTE ; // Tool State = Etat outil
    FixedLocation : BYTE ; // Fixed Location = Emplacement godet fixe
    LifetimeType : BYTE ; // Lifetime type of the Tool = Type de durée de vie
		UseFlags : BYTE ; // ? = ?
		Options : BYTE ; // ? = ?
	Smax : UDINT ; // Max Speed = Vitesse Max
	Model : UDINT ; // Tool Model = Modèle outil
		TipAngle : UDINT ; // Angle Tip = ?
	ToroidalRadius : UDINT ; // Toroidal Radius = Rayon Torique
	ChamferHeight : UDINT ; // Chamfer height = Hauteur Chanfrein
		ModelFlags : UDINT ; // ? = ?
	TeethNumber : BYTE ; // Number of Teeth = Nombre de dents
	RotationNumberCw : BYTE ; // Number of rotations clockwise = Nombre de tour sens horraire
	RotationNumberCcw : BYTE ; // Number of rotations counter-clockwise = Nombre de tour sens anti-horraire
	ThroughAirBlowTime : UINT ; // Through Air Blow Time = Temps soufflage centre outil
		ListLUserparams : ARRAY[0..3] OF DINT ;
		ListBUserparams : ARRAY [0..3] OF BYTE ;
		TailleMemByt : DINT ; 
		ListCorrecteur : ARRAY[0..44] OF DINT ; //ARRAY[0..(GV_IO.iNbrCorrTool*GV_IO.diNbrElementCorrT)-1] OF DINT; //45 correcteurs en tout dans le pire des cas 9 données *5 correcteurs
		ListCorrToolM : ARRAY[0..4] OF ST_Tool_Corrector_M ;//ARRAY[0..GV_IO.iNbrCorrTool-1] OF ST_CorrecteurM;
		ListCorrToolT : ARRAY[0..4] OF ST_Tool_Corrector_T ;
	
END_STRUCT
END_TYPE

// ---- 09_Tool_Magazine/01_DUTs/02_ST/ST_Tool_Location.TcDUT
//-----------------------------------------------------------------------------------------
//
//                  				ST_Tool_Location
//
//								Structure emplacement outil 			
//-----------------------------------------------------------------------------------------
//
//Auteur: G.GOETZ
//Création: 14.01.2026
//Dernière modification : 14.01.2026 (G.GOETZ)
//       			
//-----------------------------------------------------------------------------------------
//
//     							Liste des modifications  	
//
// 14.01.2026 (G.GOETZ) -> Création		
//-----------------------------------------------------------------------------------------

TYPE ST_Tool_Location : //140 max dont 3 bloqués 
STRUCT

	(** SETUP ENUM **)
		ePositionMag : ENUM_Position_Magazine ; // Position of the location in the Magazine : ENUM_Position_Magazine
		eToolType : ENUM_Tool_Type := ENUM_Tool_Type.Unknow ; // Type of the tool : ENUM_Tool_Type
	
	(** SETUP INT **)
		iAbsLocationNumber : INT := 0 ; // Number of the location in the Magazine
		iRelLocationNumber : INT ; // Number of the location in relative in the Magazine
		
		(* iAbsRackNumber : INT ; // Number of the rack of the location in absolute in the Magazine *)
		(* iRelRackNumber : INT ; // Number of the rack of the location in relative in the Magazine -> par exemple le numéro 3 pourrait être le 1er du magasin selon la config du projet *)
		iRackNumber : INT := 0 ; // Number of the rack of the location in the Magazine
		
		iLocationRackNumber : INT := 0 ; // Number of the location in  the rack
		
	(** SETUP FLAG **)
		bEnable : BOOL := FALSE ; // Location enable or not in the Magazine
		bForbiden : BOOL := FALSE ; // Location is forbiden or not in the Magazine
		bBlocked: BOOL := FALSE ;  // Location is blocked or not in the Magazine (because of the neighboor location have a big tool or GPS)
		bUsed : BOOL := FALSE ; // Location is used or not (defined by the User/Operator) 
		
		bBreakageOk : BOOL := FALSE ; // Breakage ctl is ok or not
		bToolPresence : BOOL := FALSE ; // Presence of the tool in the location
	
	(** PROCESS LREAL **)
		lrXcoord : LREAL := 0.0 ; // X coordinate of the location
		lrYcoord : LREAL := 0.0 ; // Y coordinate of the location
		lrZcoord : LREAL := 0.0 ; // Z coordinate of the location
	
	(** ST **)
		stToolName : ST_Tool_Name ; // Structure nom outil présent dans l'emplacement
		stToolParam : ST_Tool_Parameters ; // Structure paramètre outil présent dans l'emplacement

END_STRUCT
END_TYPE

// ---- 10_Axes/01_DUTs/01_ENUM/ENUM_Axis_Mode.TcDUT
{attribute 'qualified_only'}
{attribute 'strict'}

//-----------------------------------------------------------------------------------------
//
//                  			ENUM_Axis_Mode
//
//						Enumération des Modes des Axes			
//-----------------------------------------------------------------------------------------
//
//Auteur: G.GOETZ
//Création: 29.01.2026
//Dernière modification : 29.01.2026 (G.GOETZ)
//       			
//-----------------------------------------------------------------------------------------
//
//     							Liste des modifications  	
//
// 29.01.2026 (G.GOETZ) -> Création		
//-----------------------------------------------------------------------------------------


TYPE ENUM_Axis_Mode :
(
	Disabled := 0 , // Disable
	Manual := 1 , // Manual - Jog
	Auto := 2 , // AUTO
	Home := 3 // Home
);
END_TYPE

// ---- 10_Axes/01_DUTs/01_ENUM/ENUM_Axis_Status.TcDUT
{attribute 'qualified_only'}
{attribute 'strict'}

//-----------------------------------------------------------------------------------------
//
//                  			ENUM_Axis_Status
//
//						Enumération des Etats des Axes			
//-----------------------------------------------------------------------------------------
//
//Auteur: G.GOETZ
//Création: 29.01.2026
//Dernière modification : 29.01.2026 (G.GOETZ)
//       			
//-----------------------------------------------------------------------------------------
//
//     							Liste des modifications  	
//
// 29.01.2026 (G.GOETZ) -> Création		
//-----------------------------------------------------------------------------------------

TYPE ENUM_Axis_Status :
(
	OFF := 0 , // OFF
	Powering := 1 , // Powering in progress
	Ready := 2 , // Ready (not in movement)
	Homing := 3 , // Référencement in progress
	Jogging := 4 , // Moving in Jog	
	Autoing := 5 , // Moving in AUTO
	Error := 6 // Error
);
END_TYPE

// ---- 10_Axes/01_DUTs/01_ENUM/ENUM_Axis_Select.TcDUT
{attribute 'qualified_only'}
{attribute 'strict'}

//-----------------------------------------------------------------------------------------
//
//                  				ENUM_Axis_Select
//
//							Enumération des Axes pour choix
//-----------------------------------------------------------------------------------------
//
//Auteur: G.GOETZ
//Création: 13.01.2026
//Dernière modification : 13.01.2026 (G.GOETZ)
//       			
//-----------------------------------------------------------------------------------------
//
//     							Liste des modifications  	
//
// 13.01.2026 (G.GOETZ) -> Création		
//-----------------------------------------------------------------------------------------

TYPE ENUM_Axis_Select :
(
	None := 0 , // None Axis
	X := 1 , // X Axis
	Y := 2 , // Y Axis
	Z := 3 , // Z Axis 
	Arm := 4 // Changing Arm Axis 
);
END_TYPE

// ---- 10_Axes/01_DUTs/01_ENUM/ENUM_Handwheel_Incr_Select.TcDUT
{attribute 'qualified_only'}
{attribute 'strict'}

//-----------------------------------------------------------------------------------------
//
//                  		ENUM_Handwheel_Axis_Select
//
//				Enumération des Axes du sélecteur de la manivelle déportée			
//-----------------------------------------------------------------------------------------
//
//Auteur: G.GOETZ
//Création: 13.01.2026
//Dernière modification : 13.01.2026 (G.GOETZ)
//       			
//-----------------------------------------------------------------------------------------
//
//     							Liste des modifications  	
//
// 13.01.2026 (G.GOETZ) -> Création		
//-----------------------------------------------------------------------------------------

TYPE ENUM_Handwheel_Incr_Select :
(
	Unknow := 0 , // Unknow Speed
	x0 := 1 ,
	x1 := 2 , // Speed *1
	x10 := 3 , // Speed *10
	x100 := 4 , // Speed *100
	x1000 := 5 // Speed *1000
);
END_TYPE

// ---- 10_Axes/01_DUTs/01_ENUM/ENUM_Jog_Direction.TcDUT
{attribute 'qualified_only'}
{attribute 'strict'}

//-----------------------------------------------------------------------------------------
//
//                  				ENUM_Jog_Direction
//
//						Enumération des Direction des Axes en Jog			
//-----------------------------------------------------------------------------------------
//
//Auteur: G.GOETZ
//Création: 19.01.2026
//Dernière modification : 19.01.2026 (G.GOETZ)
//       			
//-----------------------------------------------------------------------------------------
//
//     							Liste des modifications  	
//
// 19.01.2026 (G.GOETZ) -> Création		
//-----------------------------------------------------------------------------------------

TYPE ENUM_Jog_Direction :
(
	None := 0 , // Unknow Direction
	Plus := 1 , // Positive Direction
	Minus := 2 // Negative Direction
);
END_TYPE

// ---- 10_Axes/01_DUTs/01_ENUM/ENUM_Jog_Mode.TcDUT
{attribute 'qualified_only'}
{attribute 'strict'}

//-----------------------------------------------------------------------------------------
//
//                  				ENUM_Jog_Mode
//
//						Enumération des Modes des Axes en Jog			
//-----------------------------------------------------------------------------------------
//
//Auteur: G.GOETZ
//Création: 19.01.2026
//Dernière modification : 19.01.2026 (G.GOETZ)
//       			
//-----------------------------------------------------------------------------------------
//
//     							Liste des modifications  	
//
// 19.01.2026 (G.GOETZ) -> Création		
//-----------------------------------------------------------------------------------------

TYPE ENUM_Jog_Mode :
(
	None := 0 , // Unknow Mode
	Inching := 1 , // Inching Mode = Incremental
	Continous := 2 // Continous Mode = Jog
);
END_TYPE

// ---- 10_Axes/01_DUTs/02_ST/ST_Axis.TcDUT
//-----------------------------------------------------------------------------------------
//
//                  				ST_Axis
//
//							Structure pour les Axes		
//-----------------------------------------------------------------------------------------
//
//Auteur: G.GOETZ
//Création: 29.01.2026
//Dernière modification : 29.01.2026 (G.GOETZ)
//       			
//-----------------------------------------------------------------------------------------
//
//     							Liste des modifications  	
//
// 29.01.2026 (G.GOETZ) -> Création		
//-----------------------------------------------------------------------------------------

TYPE ST_Axis :
STRUCT
	
	(** ST **)
		stDriveAx8206 : ST_Beckhoff_Drive_AX8206 ; // Structure Drive YX8206

	(** SETUP STRING **)
		strIdHMI : STRING[20] := '' ; // String for events on HMI
	
	(** SETUP INT **)
		iEventGroup : INT := 0 ; // Group for events
		iIdHMI : INT := 0 ; // Number for events on HMI
	
	(** SETUP FLAG **)
		bPresence : BOOL := FALSE ; // Presence or not
		bEventAck : BOOL := FALSE ; // Events Acknowledgement

	(** ALARMS FLAG **)
		bAlAxisFault : BOOL := FALSE ; // Axis in Fault
	
	(** PROCESS ENUM **)
		//eStatus : ENUM_Axis_Status ; // Status
		(*Jog*)
			eJogMode : TC2_MC2.E_JogMode ; // Jog Mode

	(** PROCESS LREAL **)
		(*Jog*)
			lrJogPos : LREAL ; // Jog Position
			lrJogVel : LREAL ; // Jog Velocity
			lrJogAcc : LREAL ; // Jog Acceleration
			lrJogDec : LREAL ; // Jog Decelration
			lrJogJerk : LREAL ; // Jog Jerk
		(*Auto*)
			lrAutoPosAbs : LREAL ; // AUTO Postion
			lrAutoVelAbs : LREAL ; // AUTO Velocity
			lrAutoAccAbs : LREAL ; // AUTO Acceleration
			lrAutoDecAbs : LREAL ; // AUTO Decelration
			lrAutoJerkAbs : LREAL ; // AUTO Jerk
		(*ReadParameter*)
			lrReadlrValue : LREAL ; // Read LREAL Parameter Value
			lrReadMinSoftPosLimit : LREAL ; // Read LREAL Parameter : Min Soft Limit Value
			lrReadMaxSoftPosLimit : LREAL ; // Read LREAL Parameter : Max Soft Limit Value
		(*WriteParameter*)
			lrValueMin : LREAL ; // Min Soft Limit Value for Write
			lrValueMax : LREAL ; // Max Soft Limit Value for Write
			lrWritelrValue : LREAL ; // Write LREAL Parameter Value
			
	(** PROCESS FLAG **)
		(*Power*)
			bPowerEnable : BOOL := FALSE ; // Can be Powered
		(*Stop*)
			bStopExecute : BOOL := FALSE ; // Execute a STOP
			bStopDone : BOOL ; // STOP is Done
		(*Halt*)
			bHaltExecute : BOOL := FALSE ; // Execute a HALT
			bHaltDone : BOOL ; // HALT is Done
		(*Abort*)
			bAbort : BOOL := FALSE ; // Have to Abort the mouvement
		(*Jog*)
			bJogEnable : BOOL ; // Can move in Jog
			bJogPlus : BOOL ; // Jog +
			bJogMinus : BOOL ; // Jog -
			bJogDone : BOOL ; // Jog move is done
		(*Auto*)
			bAutoEnable : BOOL ; // Can move in AUTO
			bAutoCmdAbs : BOOL ; // AUTO command
			bAutoDone : BOOL ; // AUTO move is done
		(*Reset*)
			bResetCmd : BOOL ; // Reset command
		(*Referencing*)
			bSetOffsetExecute: BOOL ; // Referencing the position at 0
			bDeleteOffsetExecute: BOOL ; // Delete the Referencing position
		(*ReadParameter*)
			bReadbEnable : BOOL ; // Read BOOL Parameter Enable
			bReadlrEnable : BOOL ; // Read LREAL Parameter Enable
			bReadbValue : BOOL ; // Read BOOL Parameter Value
			bReadbValid : BOOL ; // Read BOOL Parameter is Valid
			bReadlrValid : BOOL ; // Read LREAL Parameter is Valid
			bReadEnMinSoftPosLimit : BOOL ; // Read BOOL Parameter : Min Soft Limit Enable
			bReadEnMaxSoftPosLimit : BOOL ; // Read BOOL Parameter : Max Soft Limit Enable
		(*WriteParameter*)
			bWritebExecute : BOOL ; // Write BOOL Parameter Enable
			bWritelrExecute : BOOL ; // Write LREAL Parameter Enable
			bWritebValue : BOOL ; // Write BOOL Parameter Value
			bWritebDone : BOOL ; // Write BOOL Parameter is Done
			bWritebBusy : BOOL ; // Write BOOL Parameter is Busy
			bWritelrDone : BOOL ; // Write LREAL Parameter is Done
			bWritelrBusy : BOOL ; // Write LREAL Parameter is Busy
			
	(** MC **)
		(*ReadParameter*)
			mcAxisReadParameterb : MC_AxisParameter ; // Parameter to Read (BOOL)
			mcAxisReadParameterlr : MC_AxisParameter ; // Parameter to Read (LREAL)
		(*WriteParameter*)
			mcAxisWriteParameterb : MC_AxisParameter ; // Parameter to Write (BOOL)
			mcAxisWriteParameterlr : MC_AxisParameter ; // Parameter to Write (LREAL)
			
END_STRUCT
END_TYPE

(* Beckhoff specific parameters *) (* Index-Group 0x4000 + ID*)
(*
TYPE MC_AxisParameter : (
(* Beckhoff specific parameters *) (* Index-Group 0x4000 + ID*)
 AxisEnMinSoftPosLimit,              (* bool  *) (* IndexOffset= 16#0001_000B *)
 AxisMinSoftPosLimit,                (* lreal *) (* IndexOffset= 16#0001_000D *)
 AxisEnMaxSoftPosLimit,              (* bool  *) (* IndexOffset= 16#0001_000C *)
 AxisMaxSoftPosLimit,                (* lreal *) (* IndexOffset= 16#0001_000E *)
*)

// ---- 10_Axes/01_DUTs/02_ST/ST_Beckhoff_Drive_AX8206.TcDUT
TYPE ST_Beckhoff_Drive_AX8206 :
STRUCT
	
	// Process
	T_RESET : F_TRIG ;
	
	// Drive <=> PLC		
	AxisRef : AXIS_REF;
		
END_STRUCT
END_TYPE

// ---- 10_Axes/01_DUTs/02_ST/ST_Handwheel.TcDUT
//-----------------------------------------------------------------------------------------
//
//                  				ST_Handwheel
//
//						Structure manivelle(s) déportée(s)			
//-----------------------------------------------------------------------------------------
//
//Auteur: G.GOETZ
//Création: 19.01.2026
//Dernière modification : 19.01.2026 (G.GOETZ)
//       			
//-----------------------------------------------------------------------------------------
//
//     							Liste des modifications  	
//
// 19.01.2026 (G.GOETZ) -> Création		
//-----------------------------------------------------------------------------------------

TYPE ST_Handwheel :
STRUCT

	(** SETUP UDINT **)
		udiCounterValue : UDINT ; // Counter Value
		udiCounterValueSet : UDINT ; // Counter Value for set
	
	(** SETUP FLAG **)
		bPresence : BOOL := FALSE ; // Handwheel presence or not
		bEnable : BOOL := FALSE ; // Handwheel enable or not
		
		bAxisSelectorB0 : BOOL ; // Axis Selector Bit 0
		bAxisSelectorB1 : BOOL ; // Axis Selector Bit 1	
		bAxisSelectorB2 : BOOL ; // Axis Selector Bit 2
	
		bIncrSelectorB0 : BOOL ; // Incremental Selector Bit 0
		bIncrSelectorB1 : BOOL ; // Incremental Selector Bit 1	
		bIncrSelectorB2 : BOOL ; // Incremental Selector Bit 2	
	
		bTrackA : BOOL ; // Track A
		bTrackB : BOOL ; // Track B	
		
		bButtonPlus : BOOL ; // Button Plus
		bButtonMinus : BOOL ; // Button Minus
		bButtonFast : BOOL ; // Button Fast
	
		bCounterUnderflow : BOOL ; // Counter underflow
		bCounterOverflow : BOOL ; // Counter Overflow
		bSoftwareGateValid : BOOL ; // Counter is allowed
		bSetCounterDone : BOOL ; // Counter is Set
		bSetCounter : BOOL ; // Set Counter Value
		bSoftwareGateSet : BOOL ; // Set Counter is allowed

	(** PROCESS ENUM **)
		eAxisSelect : ENUM_Axis_Select := ENUM_Axis_Select.None ; // Axis Select
		eAxisSelectMemory : ENUM_Axis_Select := ENUM_Axis_Select.None ; // Memory of the state Axis Select
		eIncrSelect : ENUM_Handwheel_Incr_Select := ENUM_Handwheel_Incr_Select.Unknow ; // Incremental Select
		eIncrSelectMemory : ENUM_Handwheel_Incr_Select := ENUM_Handwheel_Incr_Select.Unknow ; // Memory of the state Incremental Select
		eJogDirection : ENUM_Jog_Direction := ENUM_Jog_Direction.None ; // Direction for jog
		eJogMode : ENUM_Jog_Mode := ENUM_Jog_Mode.None ; // Mode for jog	
	
	(** PROCESS REAL **)
		lrJogIncrRequest : LREAL ; // Incremental of the Jog Request
		lrJogVel : LREAL ; // Velocity for Jog in Continous Mode
	
	(** PROCESS FLAG **)	
		bPower : BOOL ; // Power
		bActivity : BOOL ; // Activity on the Handwheel
	
		bJogRequestRisingEdge : BOOL ; // Rising Edge for Jog Request	
	
END_STRUCT
END_TYPE

// ---- 11_CNC/01_DUTs/01_ENUM/ENUM_CNC_Type.TcDUT
{attribute 'qualified_only'}
{attribute 'strict'}

//-----------------------------------------------------------------------------------------
//
//                  				ENUM_CNC_Type
//
//							Enumération des types CNC			
//-----------------------------------------------------------------------------------------
//
//Auteur: G.GOETZ
//Création: 27.01.2026
//Dernière modification : 27.01.2026 (G.GOETZ)
//       			
//-----------------------------------------------------------------------------------------
//
//     							Liste des modifications  	
//
// 27.01.2026 (G.GOETZ) -> Création		
//-----------------------------------------------------------------------------------------

TYPE ENUM_CNC_Type :
(
	(*Unknow := 0 , // Unknow type*)
	Fanuc := 1 , // Fanuc CNC type
	Heidenhain := 2 // Heidenhain CNC type
);
END_TYPE

// ---- 11_CNC/01_DUTs/02_ST/ST_CNC_Fanuc_Data.TcDUT
//-----------------------------------------------------------------------------------------
//
//                  				ST_CNC_Fanuc_Data
//
//								Structure CNC_Fanuc Data 			
//-----------------------------------------------------------------------------------------
//
//Auteur: G.GOETZ
//Création: 27.01.2026
//Dernière modification : 27.01.2026 (G.GOETZ)
//       			
//-----------------------------------------------------------------------------------------
//
//     							Liste des modifications  	
//
// 27.01.2026 (G.GOETZ) -> Création		
//-----------------------------------------------------------------------------------------

TYPE ST_CNC_Fanuc_Data :
STRUCT

	(** ST **)	
		stCncMagazine : ST_CNC_Fanuc_Exchange_In_1 ; // Structure Exchange CNC -> Magazine
		stMagazineCNC : ST_CNC_Fanuc_Exchange_Out_1 ; // Structure Exchange Magzine -> CNC
		stFocasData : ST_CNC_Fanuc_Focas_Data ; // Structure for Focas data
		
	(** INT **)
		iSpindleToolLocation : INT ;
		iToolToLoadLocation : INT ;
		iSpindleToolType : INT ;
		iToolToLoadType : INT ;
		
END_STRUCT
END_TYPE

// ---- 11_CNC/01_DUTs/02_ST/ST_CNC_Fanuc_Focas_Data.TcDUT
//-----------------------------------------------------------------------------------------
//
//                  				ST_CNC_Fanuc_Focas_Data
//
//								Structure CNC_Fanuc Data 			
//-----------------------------------------------------------------------------------------
//
//Auteur: G.GOETZ
//Création: 19.02.2026
//Dernière modification : 19.02.2026 (G.GOETZ)
//       			
//-----------------------------------------------------------------------------------------
//
//     							Liste des modifications  	
//
// 19.02.2026 (G.GOETZ) -> Création		
//-----------------------------------------------------------------------------------------

TYPE ST_CNC_Fanuc_Focas_Data :
STRUCT
	
	(** ARRAY **)
	aDataReadBYTE : ARRAY [0..499] OF BYTE ;
	
	(** INT **)
	iWritingPartDataStep : INT ;
	iReadingPartDataStep : INT ;
	iWritePartDataCmd : INT ;
	iReadPartDataCmd : INT ;
	
	(** BYTE **)
	byReadIndex: BYTE ;

	(** BOOL **)
	bStartWriteDataFocas : BOOL ;	
	bStartReadDataFocas : BOOL ;

END_STRUCT
END_TYPE

// ---- 11_CNC/01_DUTs/02_ST/ST_CNC_Heidenhain_Exchange_In_1.TcDUT
//-----------------------------------------------------------------------------------------
//
//                  				ST_CNC_Heidenhain_Exchange_In
//
//								Structure Echange CNC_Heidenhain->Magasin 			
//-----------------------------------------------------------------------------------------
//
//Auteur: G.GOETZ (In agreement with ...)
//Création: 27.01.2026
//Dernière modification : 27.01.2026 (G.GOETZ)
//       			
//-----------------------------------------------------------------------------------------
//
//     							Liste des modifications  	
//
// 27.01.2026 (G.GOETZ) -> Création		
//-----------------------------------------------------------------------------------------

TYPE ST_CNC_Heidenhain_Exchange_In_1 : // 16 Bytes -> Start at X0.0 / End at X15.7 (X0.0+15.7)
STRUCT
	
	(* Byte 0 *)
		biLife : BIT ; // CNC Life bit -> X0.0
		biReserve01 : BIT ; // Reserve 01 -> X0.1
		biReserve02 : BIT ; // Reserve 02 -> X0.2
		biReserve03 : BIT ; // Reserve 03 -> X0.3
		biReserve04 : BIT ; // Reserve 04 -> X0.4
		biReserve05 : BIT ; // Reserve 05 -> X0.5
		biReserve06 : BIT ; // Reserve 06 -> X0.6
		biReserve07 : BIT ; // Reserve 07 -> X0.7

	(* Byte 1 *)
		biReserve10 : BIT ; // Reserve 10 -> X1.0
		biReserve11 : BIT ; // Reserve 11 -> X1.1
		biReserve12 : BIT ; // Reserve 12 -> X1.2
		biReserve13 : BIT ; // Reserve 13 -> X1.3
		biReserve14 : BIT ; // Reserve 14 -> X1.4
		biReserve15 : BIT ; // Reserve 15 -> X1.5
		biReserve16 : BIT ; // Reserve 16 -> X1.6
		biDoorClosed : BIT ; // CNC Door closed (operator) -> X1.7

	(* Byte 2 *)
		biReserve20 : BIT ; // Reserve 20 -> X2.0
		biReserve21 : BIT ; // Reserve 21 -> X2.1
		biReserve22 : BIT ; // Reserve 22 -> X2.2
		biReserve23 : BIT ; // Reserve 23 -> X2.3
		biReserve24 : BIT ; // Reserve 24 -> X2.4
		biReserve25 : BIT ; // Reserve 25 -> X2.5
		biReserve26 : BIT ; // Reserve 26 -> X2.6
		biReserve27 : BIT ; // Reserve 27 -> X2.7
	
	(* Byte 3 *)
		biReserve30 : BIT ; // Reserve 30 -> X3.0
		biReserve31 : BIT ; // Reserve 31 -> X3.1
		biReserve32 : BIT ; // Reserve 32 -> X3.2
		biReserve33 : BIT ; // Reserve 33 -> X3.3
		biReserve34 : BIT ; // Reserve 34 -> X3.4
		biReserve35 : BIT ; // Reserve 35 -> X3.5
		biReserve36 : BIT ; // Reserve 36 -> X3.6
		biReserve37 : BIT ; // Reserve 37 -> X3.7

	(* Byte 4-5-6-7 *)
		dwiToolSpindle : DWORD ; // Tool in CNC Spindle -> X4-5-6-7
	
	(* Byte 8-9-10-11 *)
		dwiToolToLoad : DWORD ; // Tool to Load in CNC Spindle -> X8-9-10-11
	
	(* Byte 12 *)
		byiReserve120 : BYTE ; // Reserve 120 -> X12
	
	(* Byte 13 *)
		byiReserve130 : BYTE ; // Reserve 130 -> X13
	
	(* Byte 14 *)
		byiReserve140 : BYTE ; // Reserve 140 -> X14
	
	(* Byte 15 *)
		byiReserve150 : BYTE ; // Reserve 150 -> X15
	
END_STRUCT
END_TYPE

